(* Logix 5000 project; controller CLASE_1 Emulate 5570 rev 28.11; software revision 28.02; part 12 of 15 *)
(* tags used below, declared in another part *)
   Inp_SpeedFdbk : REAL;   // Speed Feedbak in Drive Units (typ. 0-32767 = 0 to max freq.)
   Inp_Datalink : REAL;   // Auxiliary Signal (datalink) Input in Drive (raw) Units
   Inp_Ready : BOOL;   // 1=Drive is ready to run
   Inp_Running : BOOL;   // 1=Drive is Running (active)
   Inp_CommandDir : BOOL;   // 1=Drive is commanded Forward, 0=Drive is commanded Reverse
   Inp_ActualDir : BOOL;   // 1=Drive is running Forward, 0=Drive is running Reverse
   Inp_Accelerating : BOOL;   // 1=Drive is accelerating
   Inp_Decelerating : BOOL;   // 1=Drive is decelerating
   Inp_Alarm : BOOL;   // 1=Drive has an Alarm Condition (see drive display or manual)
   Inp_Faulted : BOOL;   // 1=Drive has Faulted (see drive display or manual)
   Inp_AtSpeed : BOOL;   // 1=Drive is at commanded speed
   Inp_FwdPermOK : BOOL;   // 1=Permissives OK, drive can start Forward
   Inp_FwdNBPermOK : BOOL;   // 1=Non-Bypassable Permissives OK, drive can start Forward
   Inp_RevPermOK : BOOL;   // 1=Permissives OK, drive can start Reverse
   Inp_RevNBPermOK : BOOL;   // 1=Non-Bypassable Permissives OK, motor can start Reverse
   Inp_IntlkOK : BOOL;   // 1=Interlocks OK, drive can start/run
   Inp_NBIntlkOK : BOOL;   // 1=Non-Bypassable Interlocks OK, drive can start/run
   Inp_IOFault : BOOL;   // Input Communication Status 0=OK, 1=fail
   Inp_Sim : BOOL;   // 1=Simulate working drive; 0=Start/Stop/ Monitor actual drive
   Inp_OvrdCmd : SINT;   // Override Mode Command: 0=None, 1=Stop, 2=Start Fwd 3=Start Rev
   Inp_Reset : BOOL;   // 1=Reset drive fault conditions and latched Alarms
   Cfg_HasReverse : BOOL;   // 1=Drive can be run reverse, 0=Forward only
   Cfg_AllowLocal : BOOL;   // 1=Allow Local Start/Stop without alarm, 0=Start/Stop from HMI/prog only
   Cfg_HasRunFdbk : BOOL;   // 1=Drive provides feedback signal on Inp_Running when running
   Cfg_UseRunFdbk : BOOL;   // 1=Drive run feedback should be used for failure checking
   Cfg_HasSpeedFdbk : BOOL;   // 1=Drive provides speed feedback on Inp_SpeedFdbk
   Cfg_UseSpeedFdbk : BOOL;   // 1=Drive speed determines running state, 0=state determined by drive Active input bit
   Cfg_HasInpDatalink : BOOL;   // 1=A signal is connected to Inp_Datalink
   Cfg_PCmdClear : ALIAS FOR Mode.Cfg_PCmdClear;
   Cfg_OperStopPrio : BOOL;   // 1=OCmd_Stop has priority, accepted any time, 0=OCmd_Stop only in Oper, Maint Mode.
   Cfg_OCmdResets : BOOL;   // 1=New Oper drive cmd. resets fault, 0=reset req'd to clear fault
   Cfg_OvrdPermIntlk : BOOL;   // 1=Override ignores Bypassable Perm/ Intlk; 0=always use Perm/Intlk
   Cfg_ShedOnFailToStart : BOOL;   // 1=Stop Motor and Alarm on Fail to Start; 0=Alarm only on Fail to Start
   Cfg_ShedOnIOFault : BOOL;   // 1=Stop Motor and Alarm on I/O Fault; 0=Alarm only on I/O Fault
   Cfg_SimScaleEU : BOOL;   // 1=In simulation, scale Speed Ref EU to Speed Fdbk EU
   Cfg_SimScaleRaw : BOOL;   // 1=In simulation, scale Speed Ref EU to raw, then raw to Speed Fdbk EU
   Cfg_MaxSpdRef : REAL;   // Maximum Speed Reference in EU (for limiting)
   Cfg_SpeedRefRawMin : REAL;   // Speed Reference Minimum in Drive (raw) Units (for scaling)
   Cfg_SpeedRefRawMax : REAL;   // Speed Reference Maximum in Drive (raw) Units (for scaling)
   Cfg_SpeedRefEUMin : REAL;   // Speed Reference Minimum in Engineering Units (for scaling)
   Cfg_SpeedRefEUMax : REAL;   // Speed Reference Maximum in Engineering Units (for scaling)
   Cfg_SpeedFdbkRawMin : REAL;   // Speed Feedback Minimum in Drive (raw) Units (for scaling)
   Cfg_SpeedFdbkRawMax : REAL;   // Speed Feedback Maximum in Drive (raw) Units (for scaling)
   Cfg_SpeedFdbkEUMin : REAL;   // Speed Feedback Minimum in Engineering Units (for scaling)
   Cfg_SpeedFdbkEUMax : REAL;   // Speed Feedback Maximum in Engineering Units (for scaling)
   Cfg_InpDatalinkRawMin : REAL;   // Input Datalink Minimum in Drive (raw) Units (for scaling)
   Cfg_InpDatalinkRawMax : REAL;   // Input Datalink Maximum in Drive (raw) Units (for scaling)
   Cfg_InpDatalinkEUMin : REAL;   // Input Datalink Minimum in Engineering Units (for scaling)
   Cfg_InpDatalinkEUMax : REAL;   // Input Datalink Maximum in Engineering Units (for scaling)
   Cfg_SimRampT : DINT;   // Time to ramp speed fdbk when in Simulation (sec)
   Cfg_OperKeep : SINT;   // Oper keeps control in Prog Mode: .0=Reference, .1=Start/Stop, .2=Fwd/Rev, .3=OutDatalink
   Cfg_ProgKeep : SINT;   // Prog keeps control in Oper Mode: .0=Reference, .1=Start/Stop, .2=Fwd/Rev, .3=OutDatalink
   PCmd_Start : BOOL;   // Program Command to Start Drive
   PCmd_Stop : BOOL;   // Program Command to Stop Drive
   PCmd_Fwd : BOOL;   // Program Command to set direction to Fowrard
   PCmd_Rev : BOOL;   // Program Command to set direction to Reverse
   PCmd_Reset : BOOL;   // Program Command to Reset drive fault and all Alarms requiring Reset
   PCmd_FailToStartAck : ALIAS FOR FailToStart.PCmd_Ack;   // Program Command to Acknowledge Fail to Start Alarm
   PCmd_FailToStopAck : ALIAS FOR FailToStop.PCmd_Ack;   // Program Command to Acknowledge Fail to Stop Alarm
   PCmd_IntlkTripAck : ALIAS FOR IntlkTrip.PCmd_Ack;   // Program Command to Acknowledge Interlock Trip Alarm
   PCmd_DriveFaultAck : ALIAS FOR DriveFault.PCmd_Ack;   // Program Command to Acknowledge Drive Fault Alarm
   PCmd_IOFaultAck : ALIAS FOR IOFault.PCmd_Ack;   // Program Command to Acknowledge I/O Fault Alarm
   OCmd_Start : BOOL;   // Operator Command to Start Drive
   OCmd_Stop : BOOL;   // Operator Command to Stop Drive
   OCmd_Jog : BOOL;   // Operator Command to Jog Drive (not cleared by P_VSD!)
   OCmd_Fwd : BOOL;   // Operator Command to set direction to Forward
   OCmd_Rev : BOOL;   // Operator Command to set direction to Reverse
   OCmd_Bypass : BOOL;   // Operator Command to Bypass all Bypassable Interlocks and Permissives
   OCmd_Check : BOOL;   // Operator Command to Check (not bypass) all Interlocks and Permissives
   MCmd_Disable : BOOL;   // Maintenance Command to Disable Drive
   MCmd_Enable : BOOL;   // Maintenance Command to Enable (allow to run) Drive
   OCmd_Reset : BOOL;   // Operator Command to Reset all Alarms requiring Reset
   OCmd_ResetAckAll : BOOL;   // Operator Command to Reset all Alarms and latched Shed conditions
   Out_Stop : BOOL;   // 1=Stop Drive, 0=drive left in current state
   Out_Start : BOOL;   // 1=Start Drive, 0=drive left in current state
   Out_ClearFault : BOOL;   // 1=Attempt to clear Drive Fault
   Val_SpeedFdbk : REAL;   // Speed Feedback (actual) from drive
   Val_InpDatalink : REAL;   // Input Datalink value from drive
   Val_Fdbk : SINT;   // Device Feedback 0=Stopped, 1=Running Fwd 2=Running Rev 3=Accelerating 4=Decelerating
   Sts_Starting : BOOL;   // 1=Drive requested to run and awaiting run feedback
   Sts_Running : BOOL;   // 1=Drive requested to run and is confirmed running
   Sts_CommandDir : BOOL;   // 1=Drive commanded to Forward, 0=Reverse
   Sts_ActualDir : BOOL;   // 1=Drive Actual direction is Forward, 0=Reverse
   Sts_Accel : BOOL;   // 1=Drive is Accelerating
   Sts_Decel : BOOL;   // 1=Drive is Decelerating
   Sts_NotReady : BOOL;   // 1=Drive is Not Ready (cannot be started) Check alarms, stops, faults
   Sts_Alarm : BOOL;   // 1=Drive has an Alarm (see drive display or manual)
   Sts_AtSpeed : BOOL;   // 1=Drive is running at reference speed
   Sts_Available : BOOL;   // 1=Drive available for control by automation (Prog)
   Sts_Bypass : BOOL;   // 1=Bypassable Interlocks and Permissives are Bypassed
   Sts_BypActive : BOOL;   // 1=Bypassing Active (Bypassed or Maintenance)
   Sts_Disabled : BOOL;   // 1=Drive is Disabled
   Sts_NotRdy : BOOL;   // 1=Device Not Ready, see detail bits for reason
   Nrdy_Disabled : BOOL;   // 1=Device Not Ready: Device Disabled by Maintenance
   Nrdy_CfgErr : BOOL;   // 1=Device Not Ready: Configuration Error
   Nrdy_Intlk : BOOL;   // 1=Device Not Ready: Interlock Not OK
   Nrdy_Perm : BOOL;   // 1=Device Not Ready: Permissive Not OK
   Nrdy_OperPrio : BOOL;   // 1=Device Not Ready: Operator State 0 Priority Command Requires Reset
   Nrdy_Fail : BOOL;   // 1=Device Not Ready: Device Failure (Shed Requires Reset)
   Nrdy_IOFault : BOOL;   // 1=Device Not Ready: I/O Fault (Shed Requires Reset)
   Nrdy_Trip : BOOL;   // 1=Device not Ready: Deivce Tripped (Drive Fault)
   Nrdy_DriveNR : BOOL;   // 1=Device Note Ready: Drive Not Ready
   Nrdy_NoMode : BOOL;   // 1=Device Not Ready: Device Logic Disabled / NO Mode
   Sts_MaintByp : BOOL;   // 1=A Maintenance Bypass is Active, display icon
   Sts_Err : BOOL;   // 1=Error in Config: see detail bits for reason
   Err_FdbkRaw : BOOL;   // 1=Erron in Config: Speed Fdbk Raw Min = Max
   Err_FdbkEU : BOOL;   // 1=Error in Config: Speed Fdbk EU Min = Max
   Err_RefEU : BOOL;   // 1=Error in Config: Speed Ref EU Min = Max
   Err_InpDLEU : BOOL;   // 1=Error in Config: Input Datalink EU Min = Max
   Sts_Hand : ALIAS FOR Mode.Sts_Hand;
   Sts_Maint : ALIAS FOR Mode.Sts_Maint;
   Sts_Ovrd : ALIAS FOR Mode.Sts_Ovrd;
   Sts_Prog : ALIAS FOR Mode.Sts_Prog;
   Sts_Oper : ALIAS FOR Mode.Sts_Oper;
   Sts_FailToStart : ALIAS FOR FailToStart.Inp;   // 1=Drive Failed to Start (One-Shot)
   Sts_FailToStop : ALIAS FOR FailToStop.Inp;   // 1=Drive Failed to Stop
   Sts_IntlkTrip : ALIAS FOR IntlkTrip.Inp;   // 1=Drive was stopped by an Interlock NOT OK (One-Shot)
   Sts_DriveFault : ALIAS FOR DriveFault.Inp;   // 1=Drive Fault (see drive display or manual)
   Sts_IOFault : ALIAS FOR IOFault.Inp;   // I/O Comm Fault Status (0=OK, 1=Bad)
   Rdy_Fwd : BOOL;   // 1=Ready to receive OCmd_Fwd (enabled HMI button)
   Rdy_Rev : BOOL;   // 1=Ready to receive OCmd_Rev (enables HMI button)
   Rdy_Bypass : BOOL;   // 1=Ready to receive OCmd_Bypass (enables HMI button)
   Rdy_Check : BOOL;   // 1=Ready to receive OCmd_Check (enables HMI button)
   Rdy_Disable : BOOL;   // 1=Ready to receive MCmd_Disable (enables HMI button)
   Rdy_Enable : BOOL;   // 1=Ready to receive MCmd_Enable (enables HMI button)
   P_VSD : BOOL;   // Unique Parameter Name for auto - discovery
   Mode : P_Mode;   // Drive Mode Selection
   IOFault : P_Alarm;   // I/O Fault Alarm
   IntlkTrip : P_Alarm;   // Interlock Trip Alarm
   FailToStop : P_Alarm;   // Drive Failed to Stop Alarm
   FailToStart : P_Alarm;   // Drive Failed to Start Alarm
   Wrk_Run : BOOL;   // 1=Drive should be "running", 0=should be "stopped"
   Wrk_StartRetrigT : TIMER;   // Time to pulse start output on start command retrigger (Maint)
   Wrk_StopRetrigT : TIMER;   // Time to pulse stop output on stop command retrigger (Maint)
   Wrk_RunFdbk : BOOL;   // Run Feedback based on mode, simulation, etc. 1=running
   Wrk_Bypass : BOOL;   // Internal Bypassable Permissives and Interlocks are Bypassed flag
   Wrk_Disabled : BOOL;   // Internal Drive is Disabled
   DriveFault : P_Alarm;   // Drive Faulted Alarm
   Wrk_SpeedRef : REAL;   // Working copy of Speed Reference (for limiting)
   Wrk_Rev : BOOL;   // Working (internal) Direction 1=Reverse 0=Forward (default)
   Wrk_Jog : BOOL;   // 1=Jog Drive, 0=Drive not jogging
   Wrk_ResetT : TIMER;   // Reset Output Pulse Timer
   Wrk_ResetONS : BOOL;   // One-Shot to fire Reset Timer to ensure min. output ON time.
   Wrk_StopT : TIMER;   // Stop Check Timer (for Fail to Stop)
   Wrk_StartT : TIMER;   // Start Check Timer (for Fail to Start)
   Wrk_Retrigger : BOOL;   // Maint Start issued while running or Stop while stopped
   Wrk_Step : REAL;   // Amount to change simulated Speed Fdbk this scan (ramp)
   Wrk_ScanTime : REAL;   // Seconds since previous scan
   Wrk_SimFdbkTgt : REAL;   // Speed Ref converted to Speed Fdbk units for simulation: target speed fdbk
   Wrk_JogT : TIMER;   // Jog Timer
   Wrk_SimScaleEUONS : BOOL;   // Cfg_SimScaleEU became true this scan
   Wrk_SimScaleRawONS : BOOL;   // Cfg_SimScaleRaw became true this scan
   Wrk_NotRdyONS : BOOL;   // Assert Stop on One-Shot of Sts_NotRdy
   Wrk_NotRdy : BOOL;   // Device Not Ready conditions excluding shed latches
   Wrk_StartInhT : TIMER;   // Local Start Inhibit Timer
   Wrk_StopInhT : TIMER;   // Local Stop Inhibit Timer
   Wrk_Hand : BOOL;   // Perform Hand Mode alignment with actual device state
   Wrk_RevCmdRcvd : BOOL;   // A Reverse direction command was received this scan.
   Wrk_FwdCmdRcvd : BOOL;   // A Forward direction command was received this scan
(* P_VSD, continued *)

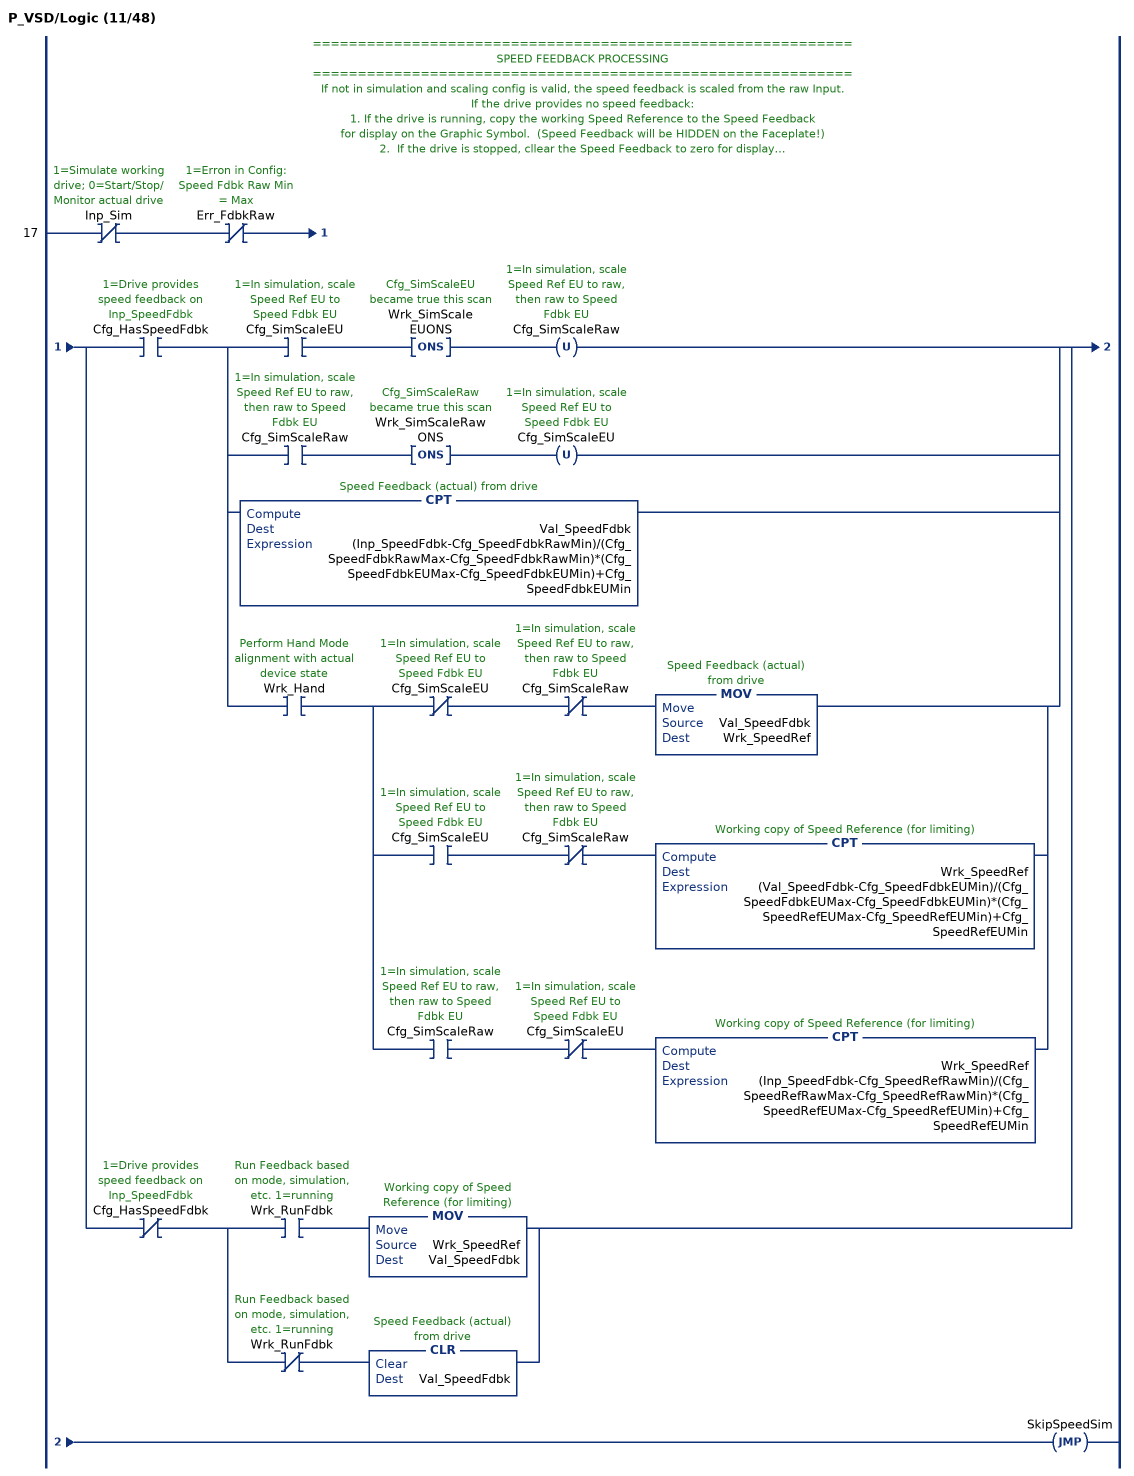
   // ============================================================
   // SPEED FEEDBACK PROCESSING
   // ============================================================
   // If not in simulation and scaling config is valid, the speed feedback is scaled from the raw Input.
   // If the drive provides no speed feedback:
   // 1. If the drive is running, copy the working Speed Reference to the Speed Feedback
   // for display on the Graphic Symbol.  (Speed Feedback will be HIDDEN on the Faceplate!)
   // 2.  If the drive is stopped, cllear the Speed Feedback to zero for display.
   // #####  V3.0-00  2013-06-30:  Added Cfg_HasSpeedFdbk  #####
   // #####  V3.0-05  2014-05-20:  Modified to prevent both Simulation  #####
   // #####  scaling bits from being set at the same time.  #####
   // #####  V3.1-04 Patch01  2015-09-25:  Added logic for Cfg_HasSpeedFdbk = 0  #####
   // #####  V3.5-04  2016-09-30:  Modified to ensure instruction  #####
   // #####  aligns with actual state of the drive on transistion from Sim to Real.  #####
   17: XIO(Inp_Sim)XIO(Err_FdbkRaw)[XIC(Cfg_HasSpeedFdbk) [XIC(Cfg_SimScaleEU) ONS(Wrk_SimScaleEUONS) OTU(Cfg_SimScaleRaw) ,XIC(Cfg_SimScaleRaw) ONS(Wrk_SimScaleRawONS) OTU(Cfg_SimScaleEU) ,CPT(Val_SpeedFdbk,(Inp_SpeedFdbk-Cfg_SpeedFdbkRawMin)/(Cfg_SpeedFdbkRawMax-Cfg_SpeedFdbkRawMin)*(Cfg_SpeedFdbkEUMax-Cfg_SpeedFdbkEUMin)+Cfg_SpeedFdbkEUMin) ,XIC(Wrk_Hand) [XIO(Cfg_SimScaleEU) XIO(Cfg_SimScaleRaw) MOV(Val_SpeedFdbk,Wrk_SpeedRef) ,XIC(Cfg_SimScaleEU) XIO(Cfg_SimScaleRaw) CPT(Wrk_SpeedRef,(Val_SpeedFdbk-Cfg_SpeedFdbkEUMin)/(Cfg_SpeedFdbkEUMax-Cfg_SpeedFdbkEUMin)*(Cfg_SpeedRefEUMax-Cfg_SpeedRefEUMin)+Cfg_SpeedRefEUMin) ,XIC(Cfg_SimScaleRaw) XIO(Cfg_SimScaleEU) CPT(Wrk_SpeedRef,(Inp_SpeedFdbk-Cfg_SpeedRefRawMin)/(Cfg_SpeedRefRawMax-Cfg_SpeedRefRawMin)*(Cfg_SpeedRefEUMax-Cfg_SpeedRefEUMin)+Cfg_SpeedRefEUMin) ] ] ,XIO(Cfg_HasSpeedFdbk) [XIC(Wrk_RunFdbk) MOV(Wrk_SpeedRef,Val_SpeedFdbk) ,XIO(Wrk_RunFdbk) CLR(Val_SpeedFdbk) ] ]JMP(SkipSpeedSim);
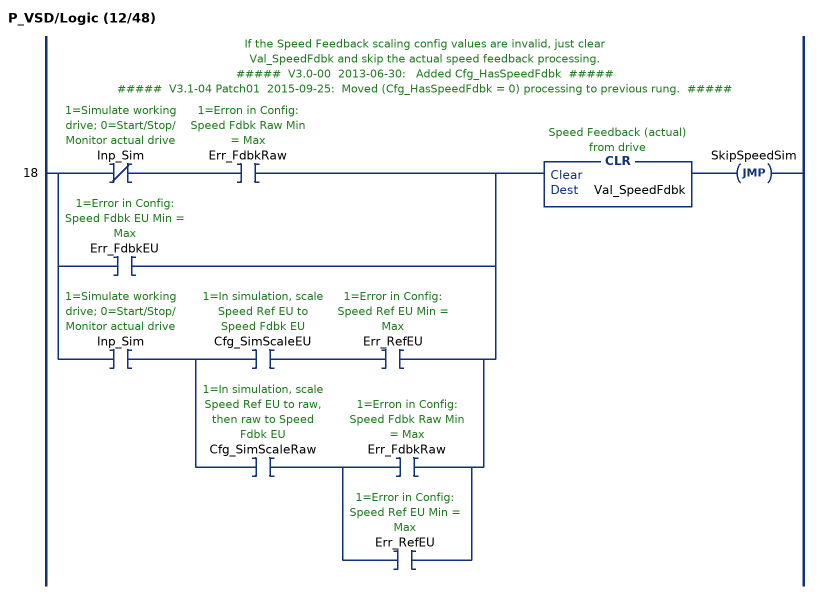
   // If the Speed Feedback scaling config values are invalid, just clear
   // Val_SpeedFdbk and skip the actual speed feedback processing.
   // #####  V3.0-00  2013-06-30:   Added Cfg_HasSpeedFdbk  #####
   // #####  V3.1-04 Patch01  2015-09-25:  Moved (Cfg_HasSpeedFdbk = 0) processing to previous rung.  #####
   18: [XIO(Inp_Sim) XIC(Err_FdbkRaw) ,XIC(Err_FdbkEU) ,XIC(Inp_Sim) [XIC(Cfg_SimScaleEU) XIC(Err_RefEU) ,XIC(Cfg_SimScaleRaw) [XIC(Err_FdbkRaw) ,XIC(Err_RefEU) ] ] ]CLR(Val_SpeedFdbk)JMP(SkipSpeedSim);
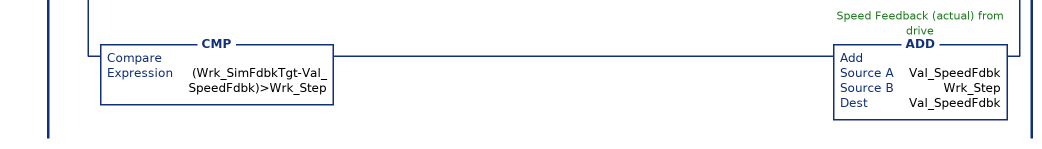
   // If in simulation, simulate accel/decel.
   19: XIC(Inp_Sim)[[XIC(Wrk_Run) ,XIC(Wrk_Jog) ] [XIO(Cfg_SimScaleEU) XIO(Cfg_SimScaleRaw) MOV(Wrk_SpeedRef,Wrk_SimFdbkTgt) ,[XIC(Cfg_SimScaleEU) XIO(Cfg_SimScaleRaw) CPT(Wrk_SimFdbkTgt,(Wrk_SpeedRef-Cfg_SpeedRefEUMin)/(Cfg_SpeedRefEUMax-Cfg_SpeedRefEUMin)*(Cfg_SpeedFdbkEUMax-Cfg_SpeedFdbkEUMin)+Cfg_SpeedFdbkEUMin) ,XIC(Cfg_SimScaleRaw) [CPT(Wrk_SimFdbkTgt,(Wrk_SpeedRef-Cfg_SpeedRefEUMin)/(Cfg_SpeedRefEUMax-Cfg_SpeedRefEUMin)*(Cfg_SpeedRefRawMax-Cfg_SpeedRefRawMin)+Cfg_SpeedRefRawMin) ,CPT(Wrk_SimFdbkTgt,(Wrk_SimFdbkTgt-Cfg_SpeedFdbkRawMin)/(Cfg_SpeedFdbkRawMax-Cfg_SpeedFdbkRawMin)*(Cfg_SpeedFdbkEUMax-Cfg_SpeedFdbkEUMin)+Cfg_SpeedFdbkEUMin) ] ] ] ,[XIO(Wrk_Run) XIO(Wrk_Jog) ,XIO(Wrk_Rev) XIO(Sts_ActualDir) ,XIC(Wrk_Rev) XIC(Sts_ActualDir) ] CLR(Wrk_SimFdbkTgt) ,GRT(Cfg_SimRampT,0) [CPT(Wrk_Step,Cfg_MaxSpdRef/Cfg_SimRampT*Wrk_ScanTime) ,XIC(Cfg_SimScaleEU) XIO(Cfg_SimScaleRaw) CPT(Wrk_Step,(Wrk_Step-Cfg_SpeedRefEUMin)/(Cfg_SpeedRefEUMax-Cfg_SpeedRefEUMin)*(Cfg_SpeedFdbkEUMax-Cfg_SpeedFdbkEUMin)+Cfg_SpeedFdbkEUMin) ,XIC(Cfg_SimScaleRaw) [CPT(Wrk_Step,(Wrk_Step-Cfg_SpeedRefEUMin)/(Cfg_SpeedRefEUMax-Cfg_SpeedRefEUMin)*(Cfg_SpeedRefRawMax-Cfg_SpeedRefRawMin)+Cfg_SpeedRefRawMin) ,CPT(Wrk_Step,(Wrk_Step-Cfg_SpeedFdbkRawMin)/(Cfg_SpeedFdbkRawMax-Cfg_SpeedFdbkRawMin)*(Cfg_SpeedFdbkEUMax-Cfg_SpeedFdbkEUMin)+Cfg_SpeedFdbkEUMin) ] ] ,LEQ(Cfg_SimRampT,0) MOV(1.50000000e+038,Wrk_Step) ,CMP(ABS(Val_SpeedFdbk-Wrk_SimFdbkTgt)<=Wrk_Step) MOV(Wrk_SimFdbkTgt,Val_SpeedFdbk) ,CMP((Val_SpeedFdbk-Wrk_SimFdbkTgt)>Wrk_Step) SUB(Val_SpeedFdbk,Wrk_Step,Val_SpeedFdbk) ,CMP((Wrk_SimFdbkTgt-Val_SpeedFdbk)>Wrk_Step) ADD(Val_SpeedFdbk,Wrk_Step,Val_SpeedFdbk) ];
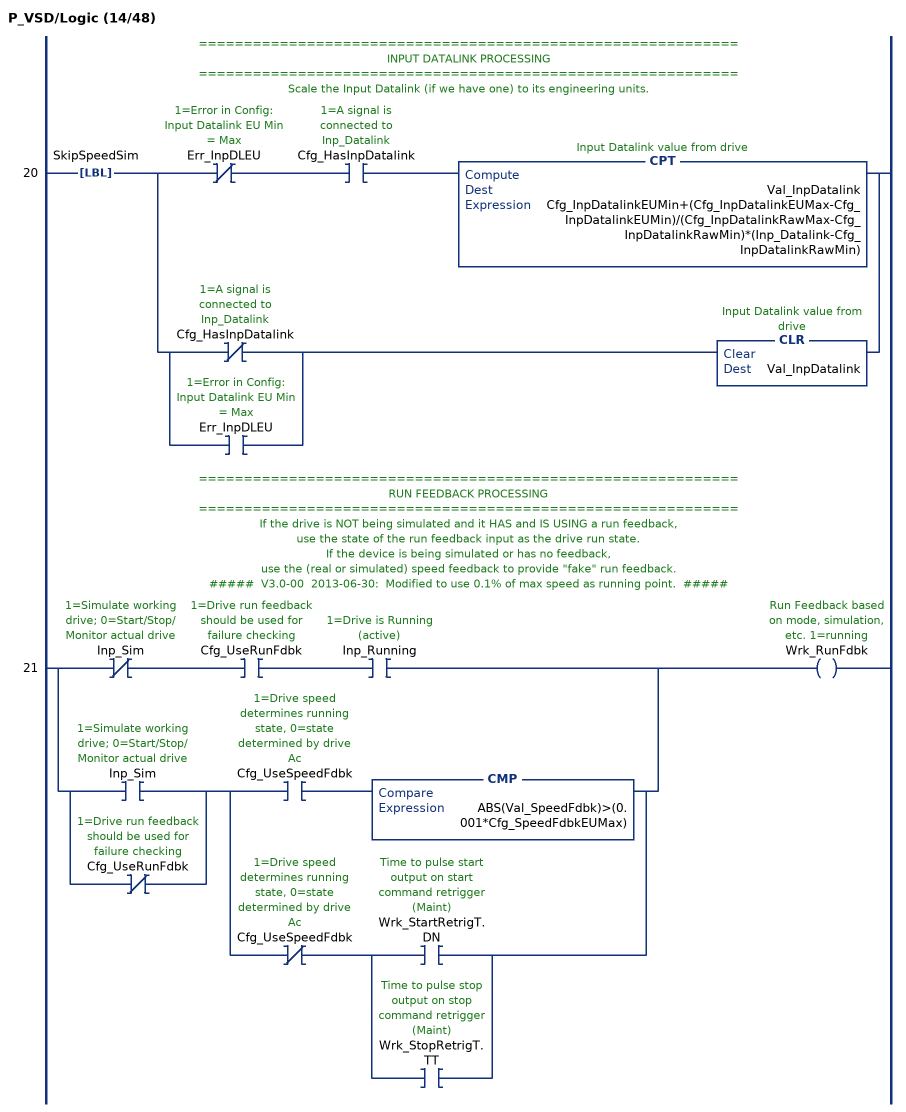
   // ============================================================
   // INPUT DATALINK PROCESSING
   // ============================================================
   // Scale the Input Datalink (if we have one) to its engineering units.
   20: LBL(SkipSpeedSim)[XIO(Err_InpDLEU) XIC(Cfg_HasInpDatalink) CPT(Val_InpDatalink,Cfg_InpDatalinkEUMin+(Cfg_InpDatalinkEUMax-Cfg_InpDatalinkEUMin)/(Cfg_InpDatalinkRawMax-Cfg_InpDatalinkRawMin)*(Inp_Datalink-Cfg_InpDatalinkRawMin)) ,[XIO(Cfg_HasInpDatalink) ,XIC(Err_InpDLEU) ] CLR(Val_InpDatalink) ];
   // ============================================================
   // RUN FEEDBACK PROCESSING
   // ============================================================
   // If the drive is NOT being simulated and it HAS and IS USING a run feedback,
   // use the state of the run feedback input as the drive run state.
   // If the device is being simulated or has no feedback,
   // use the (real or simulated) speed feedback to provide "fake" run feedback.
   // #####  V3.0-00  2013-06-30:  Modified to use 0.1% of max speed as running point.  #####
   21: [XIO(Inp_Sim) XIC(Cfg_UseRunFdbk) XIC(Inp_Running) ,[XIC(Inp_Sim) ,XIO(Cfg_UseRunFdbk) ] [XIC(Cfg_UseSpeedFdbk) CMP(ABS(Val_SpeedFdbk)>(0.001*Cfg_SpeedFdbkEUMax)) ,XIO(Cfg_UseSpeedFdbk) [XIC(Wrk_StartRetrigT.DN) ,XIC(Wrk_StopRetrigT.TT) ] ] ]OTE(Wrk_RunFdbk);
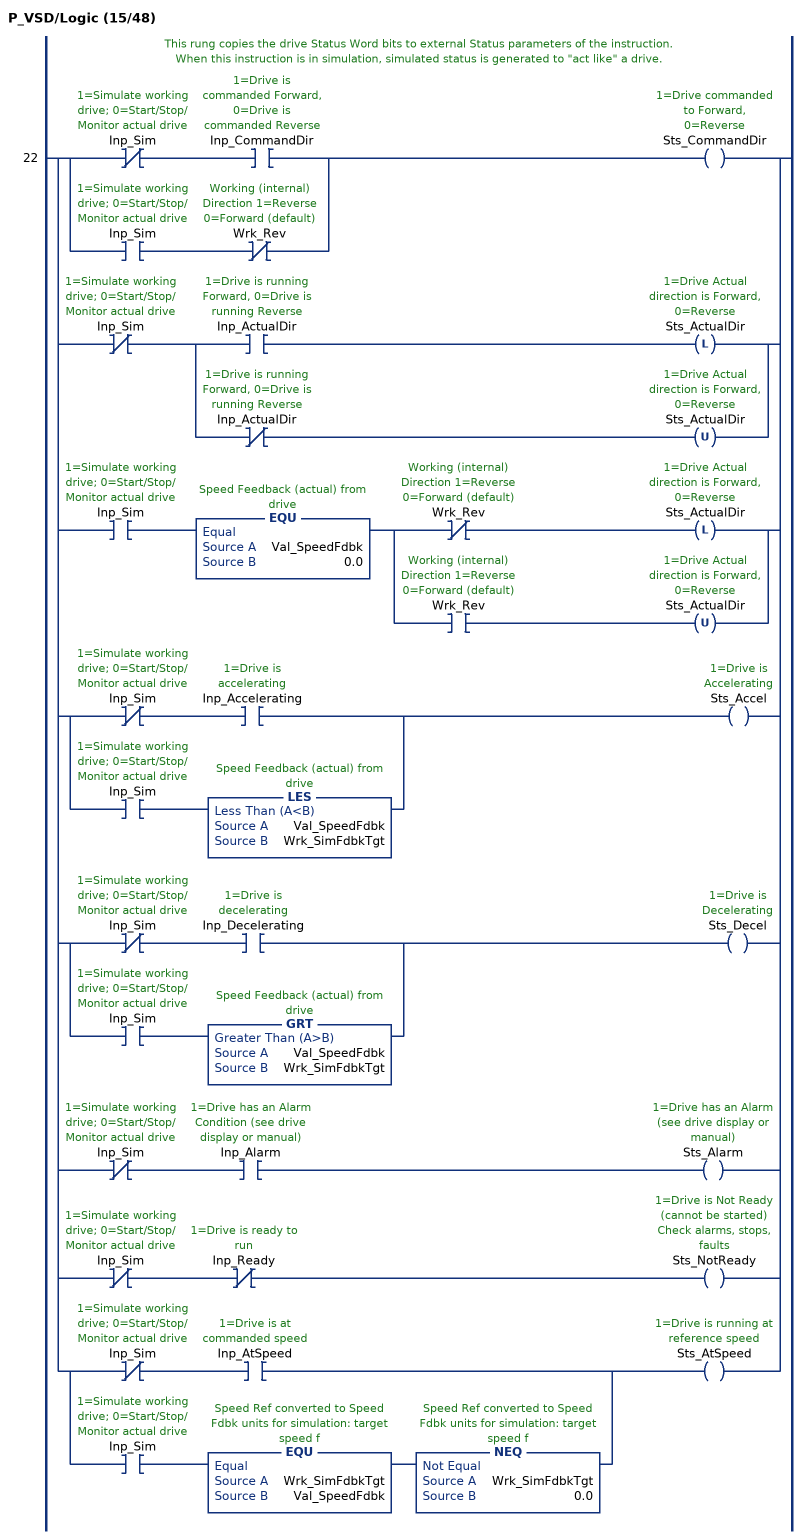
   // This rung copies the drive Status Word bits to external Status parameters of the instruction.
   // When this instruction is in simulation, simulated status is generated to "act like" a drive.
   22: [[XIO(Inp_Sim) XIC(Inp_CommandDir) ,XIC(Inp_Sim) XIO(Wrk_Rev) ] OTE(Sts_CommandDir) ,[XIO(Inp_Sim) [XIC(Inp_ActualDir) OTL(Sts_ActualDir) ,XIO(Inp_ActualDir) OTU(Sts_ActualDir) ] ,XIC(Inp_Sim) EQU(Val_SpeedFdbk,0.0) [XIO(Wrk_Rev) OTL(Sts_ActualDir) ,XIC(Wrk_Rev) OTU(Sts_ActualDir) ] ] ,[XIO(Inp_Sim) XIC(Inp_Accelerating) ,XIC(Inp_Sim) LES(Val_SpeedFdbk,Wrk_SimFdbkTgt) ] OTE(Sts_Accel) ,[XIO(Inp_Sim) XIC(Inp_Decelerating) ,XIC(Inp_Sim) GRT(Val_SpeedFdbk,Wrk_SimFdbkTgt) ] OTE(Sts_Decel) ,XIO(Inp_Sim) XIC(Inp_Alarm) OTE(Sts_Alarm) ,XIO(Inp_Sim) XIO(Inp_Ready) OTE(Sts_NotReady) ,[XIO(Inp_Sim) XIC(Inp_AtSpeed) ,XIC(Inp_Sim) EQU(Wrk_SimFdbkTgt,Val_SpeedFdbk) NEQ(Wrk_SimFdbkTgt,0.0) ] OTE(Sts_AtSpeed) ];
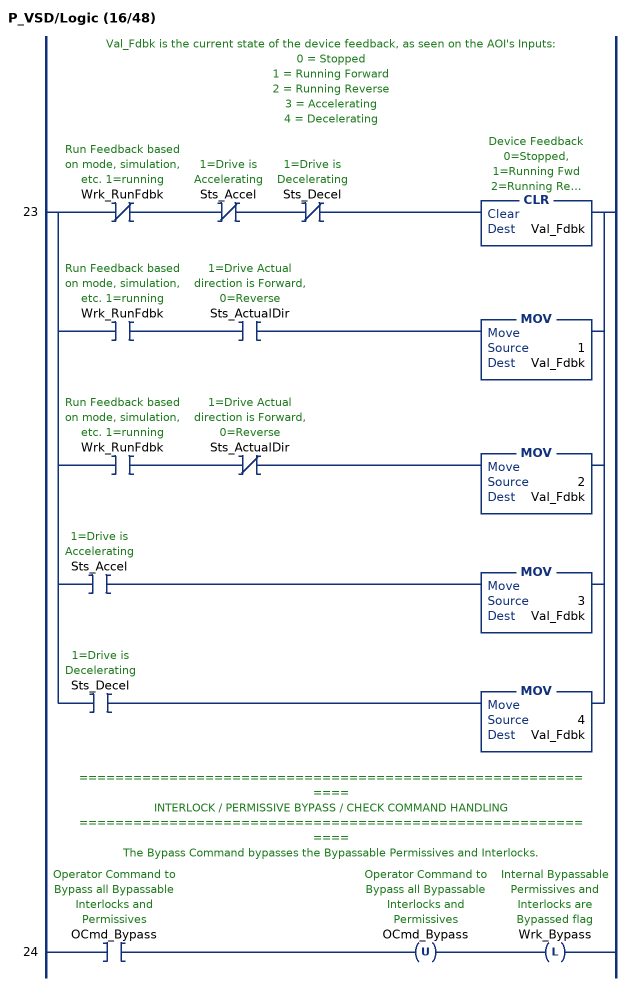
   // Val_Fdbk is the current state of the device feedback, as seen on the AOI's Inputs:
   // 0 = Stopped
   // 1 = Running Forward
   // 2 = Running Reverse
   // 3 = Accelerating
   // 4 = Decelerating
   23: [XIO(Wrk_RunFdbk) XIO(Sts_Accel) XIO(Sts_Decel) CLR(Val_Fdbk) ,XIC(Wrk_RunFdbk) XIC(Sts_ActualDir) MOV(1,Val_Fdbk) ,XIC(Wrk_RunFdbk) XIO(Sts_ActualDir) MOV(2,Val_Fdbk) ,XIC(Sts_Accel) MOV(3,Val_Fdbk) ,XIC(Sts_Decel) MOV(4,Val_Fdbk) ];
   // ============================================================
   // INTERLOCK / PERMISSIVE BYPASS / CHECK COMMAND HANDLING
   // ============================================================
   // The Bypass Command bypasses the Bypassable Permissives and Interlocks.
   24: XIC(OCmd_Bypass)OTU(OCmd_Bypass)OTL(Wrk_Bypass);
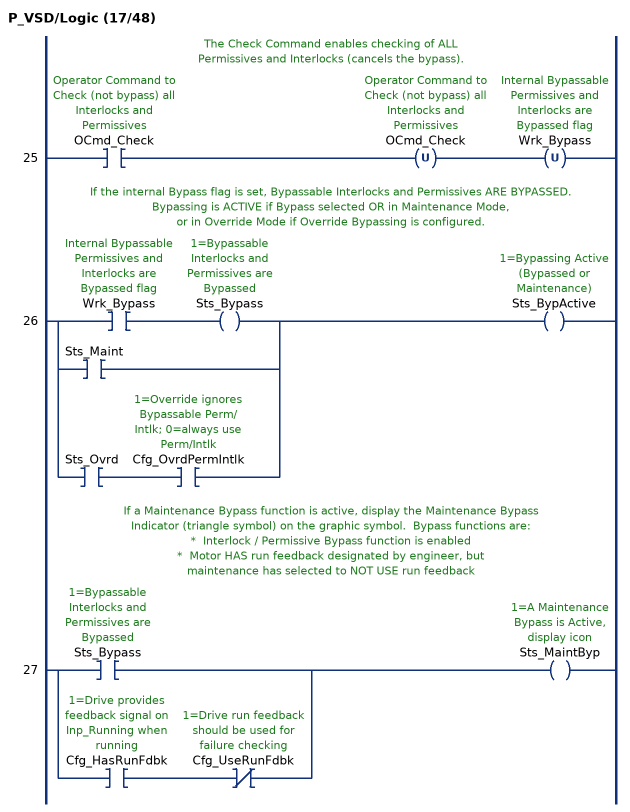
   // The Check Command enables checking of ALL
   // Permissives and Interlocks (cancels the bypass).
   25: XIC(OCmd_Check)OTU(OCmd_Check)OTU(Wrk_Bypass);
   // If the internal Bypass flag is set, Bypassable Interlocks and Permissives ARE BYPASSED.
   // Bypassing is ACTIVE if Bypass selected OR in Maintenance Mode,
   // or in Override Mode if Override Bypassing is configured.
   26: [XIC(Wrk_Bypass) OTE(Sts_Bypass) ,XIC(Sts_Maint) ,XIC(Sts_Ovrd) XIC(Cfg_OvrdPermIntlk) ]OTE(Sts_BypActive);
   // If a Maintenance Bypass function is active, display the Maintenance Bypass
   // Indicator (triangle symbol) on the graphic symbol.  Bypass functions are:
   // *  Interlock / Permissive Bypass function is enabled
   // *  Motor HAS run feedback designated by engineer, but
   // maintenance has selected to NOT USE run feedback
   27: [XIC(Sts_Bypass) ,XIC(Cfg_HasRunFdbk) XIO(Cfg_UseRunFdbk) ]OTE(Sts_MaintByp);
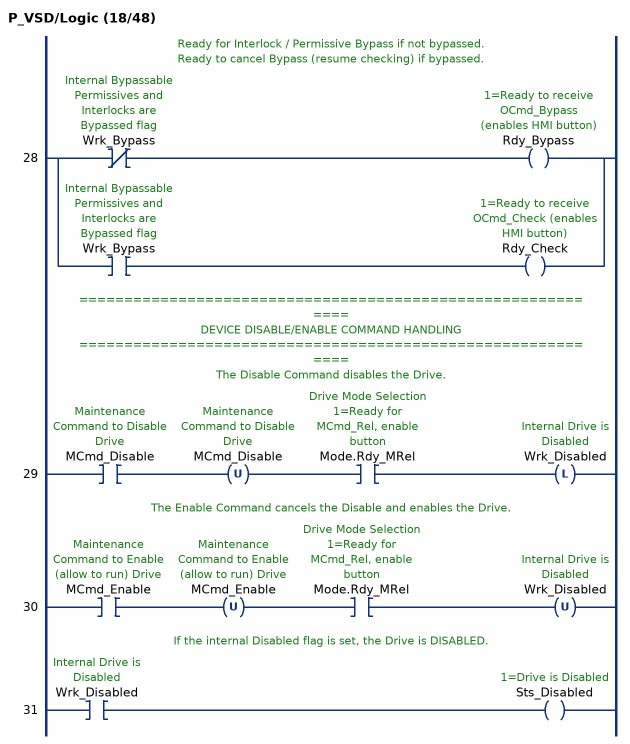
   // Ready for Interlock / Permissive Bypass if not bypassed.
   // Ready to cancel Bypass (resume checking) if bypassed.
   28: [XIO(Wrk_Bypass) OTE(Rdy_Bypass) ,XIC(Wrk_Bypass) OTE(Rdy_Check) ];
   // ============================================================
   // DEVICE DISABLE/ENABLE COMMAND HANDLING
   // ============================================================
   // The Disable Command disables the Drive.
   29: XIC(MCmd_Disable)OTU(MCmd_Disable)XIC(Mode.Rdy_MRel)OTL(Wrk_Disabled);
   // The Enable Command cancels the Disable and enables the Drive.
   30: XIC(MCmd_Enable)OTU(MCmd_Enable)XIC(Mode.Rdy_MRel)OTU(Wrk_Disabled);
   // If the internal Disabled flag is set, the Drive is DISABLED.
   31: XIC(Wrk_Disabled)OTE(Sts_Disabled);
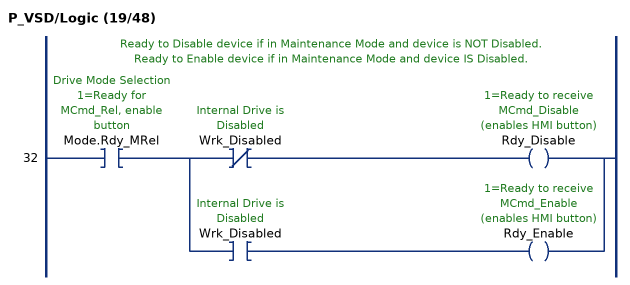
   // Ready to Disable device if in Maintenance Mode and device is NOT Disabled.
   // Ready to Enable device if in Maintenance Mode and device IS Disabled.
   32: XIC(Mode.Rdy_MRel)[XIO(Wrk_Disabled) OTE(Rdy_Disable) ,XIC(Wrk_Disabled) OTE(Rdy_Enable) ];
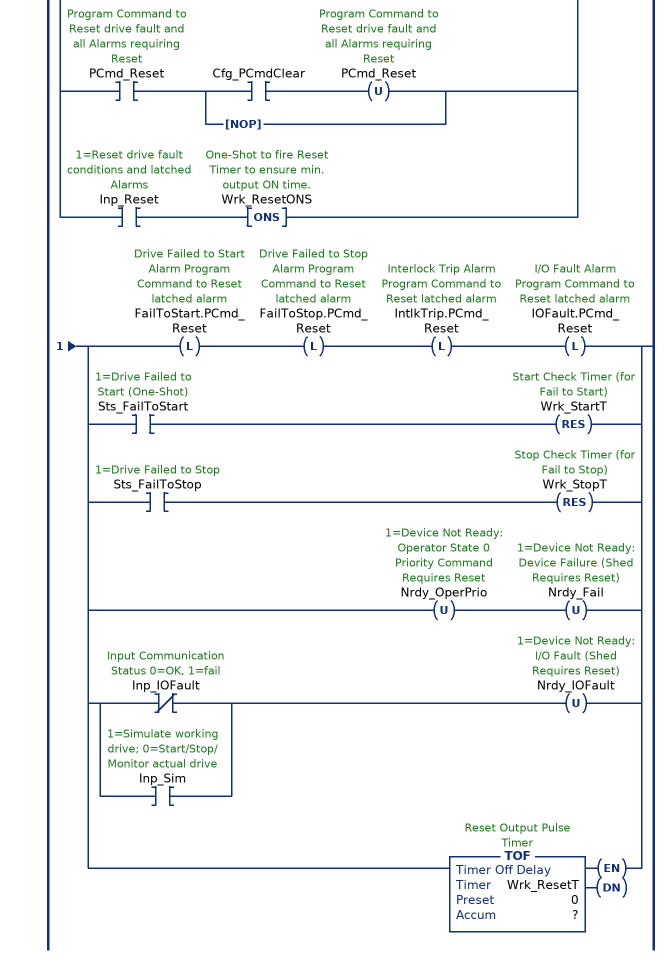
   // ============================================================
   // ALARM RESET COMMAND HANDLING
   // ============================================================
   // This rung handles the Alarm Reset Input and Commands
   // and the "Reset and Ack All" Operator Command.
   // This rung processes received Reset Commands from:
   // 1.  The Operator via HMI Operator Command, or
   // 2.  Higher-level strategies via Program Command
   // 3.  Pushbuttons or other block via Input
   // 4.  Resets initiated by other device Operator Commands (if configured to do so)
   // and forwards the Reset to ALL Alarms and latched Shed conditions.
   // The reset starts the Reset Timer (One-Shot Off-Delay)
   // to ensure the output is held on for at least the minimum time.
   // #####  V3.1-00  2014-06-30: Added Not Ready reason bits (Nrdy_xxx)  #####
   // #####  V3.1-01  2014-08-29:  Corrections to Nrdy_ trip and reset logic.  #####
   33: [XIC(OCmd_Reset) OTU(OCmd_Reset) ,[XIC(OCmd_Start) ,XIC(OCmd_Jog) ,XIC(OCmd_Stop) ] XIC(Cfg_OCmdResets) [XIC(Sts_Oper) XIO(Cfg_ProgKeep.1) ,XIC(Sts_Maint) ,XIC(Sts_Prog) XIC(Cfg_OperKeep.1) ] ,XIC(OCmd_ResetAckAll) OTU(OCmd_ResetAckAll) [OTL(PCmd_FailToStartAck) ,OTL(PCmd_FailToStopAck) ,OTL(PCmd_DriveFaultAck) ,OTL(PCmd_IntlkTripAck) ,OTL(PCmd_IOFaultAck) ] ,XIC(PCmd_Reset) [XIC(Cfg_PCmdClear) OTU(PCmd_Reset) ,NOP() ] ,XIC(Inp_Reset) ONS(Wrk_ResetONS) ][OTL(FailToStart.PCmd_Reset) OTL(FailToStop.PCmd_Reset) OTL(IntlkTrip.PCmd_Reset) OTL(IOFault.PCmd_Reset) ,XIC(Sts_FailToStart) RES(Wrk_StartT) ,XIC(Sts_FailToStop) RES(Wrk_StopT) ,OTU(Nrdy_OperPrio) OTU(Nrdy_Fail) ,[XIO(Inp_IOFault) ,XIC(Inp_Sim) ] OTU(Nrdy_IOFault) ,TOF(Wrk_ResetT,?,?) ];
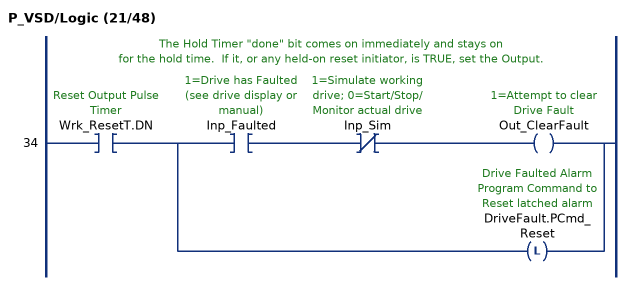
   // The Hold Timer "done" bit comes on immediately and stays on
   // for the hold time.  If it, or any held-on reset initiator, is TRUE, set the Output.
   34: XIC(Wrk_ResetT.DN)[XIC(Inp_Faulted) XIO(Inp_Sim) OTE(Out_ClearFault) ,OTL(DriveFault.PCmd_Reset) ];
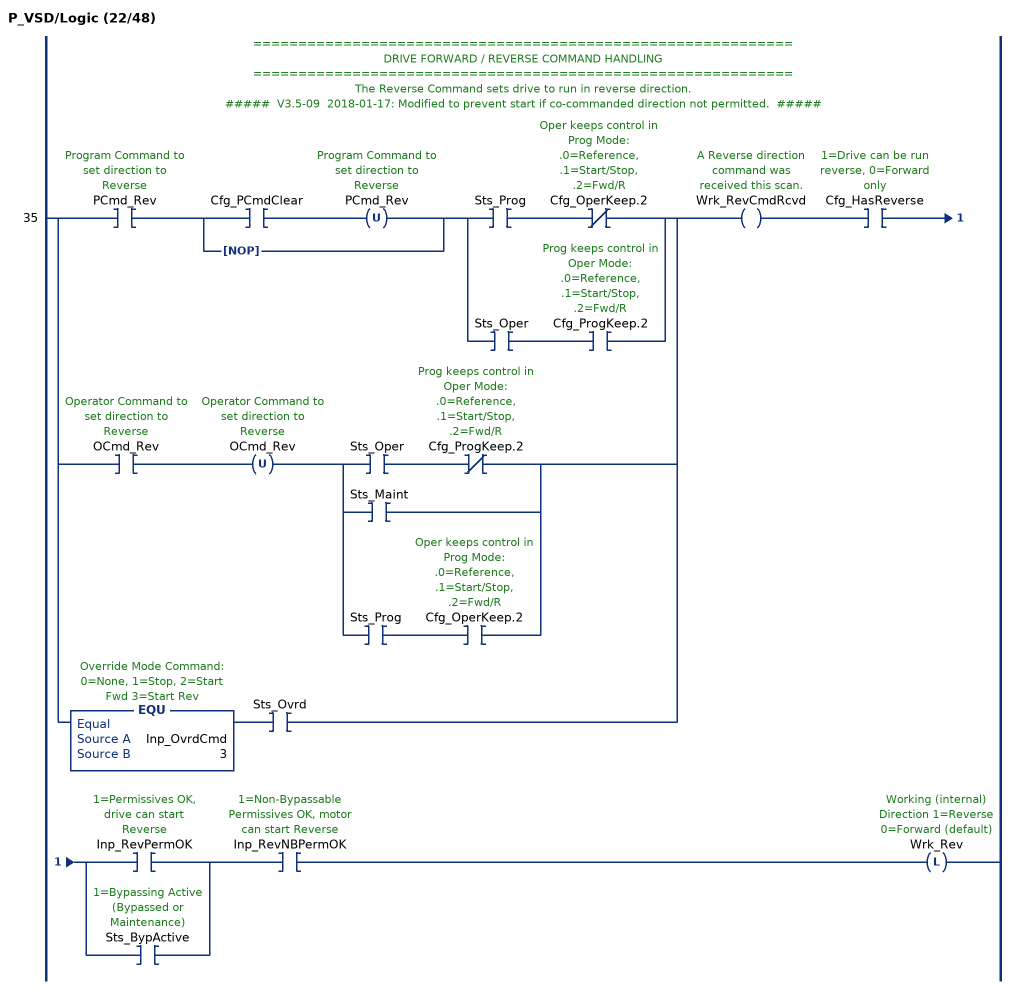
   // ============================================================
   // DRIVE FORWARD / REVERSE COMMAND HANDLING
   // ============================================================
   // The Reverse Command sets drive to run in reverse direction.
   // #####  V3.5-09  2018-01-17: Modified to prevent start if co-commanded direction not permitted.  #####
   35: [XIC(PCmd_Rev) [XIC(Cfg_PCmdClear) OTU(PCmd_Rev) ,NOP() ] [XIC(Sts_Prog) XIO(Cfg_OperKeep.2) ,XIC(Sts_Oper) XIC(Cfg_ProgKeep.2) ] ,XIC(OCmd_Rev) OTU(OCmd_Rev) [XIC(Sts_Oper) XIO(Cfg_ProgKeep.2) ,XIC(Sts_Maint) ,XIC(Sts_Prog) XIC(Cfg_OperKeep.2) ] ,EQU(Inp_OvrdCmd,3) XIC(Sts_Ovrd) ]OTE(Wrk_RevCmdRcvd)XIC(Cfg_HasReverse)[XIC(Inp_RevPermOK) ,XIC(Sts_BypActive) ]XIC(Inp_RevNBPermOK)OTL(Wrk_Rev);
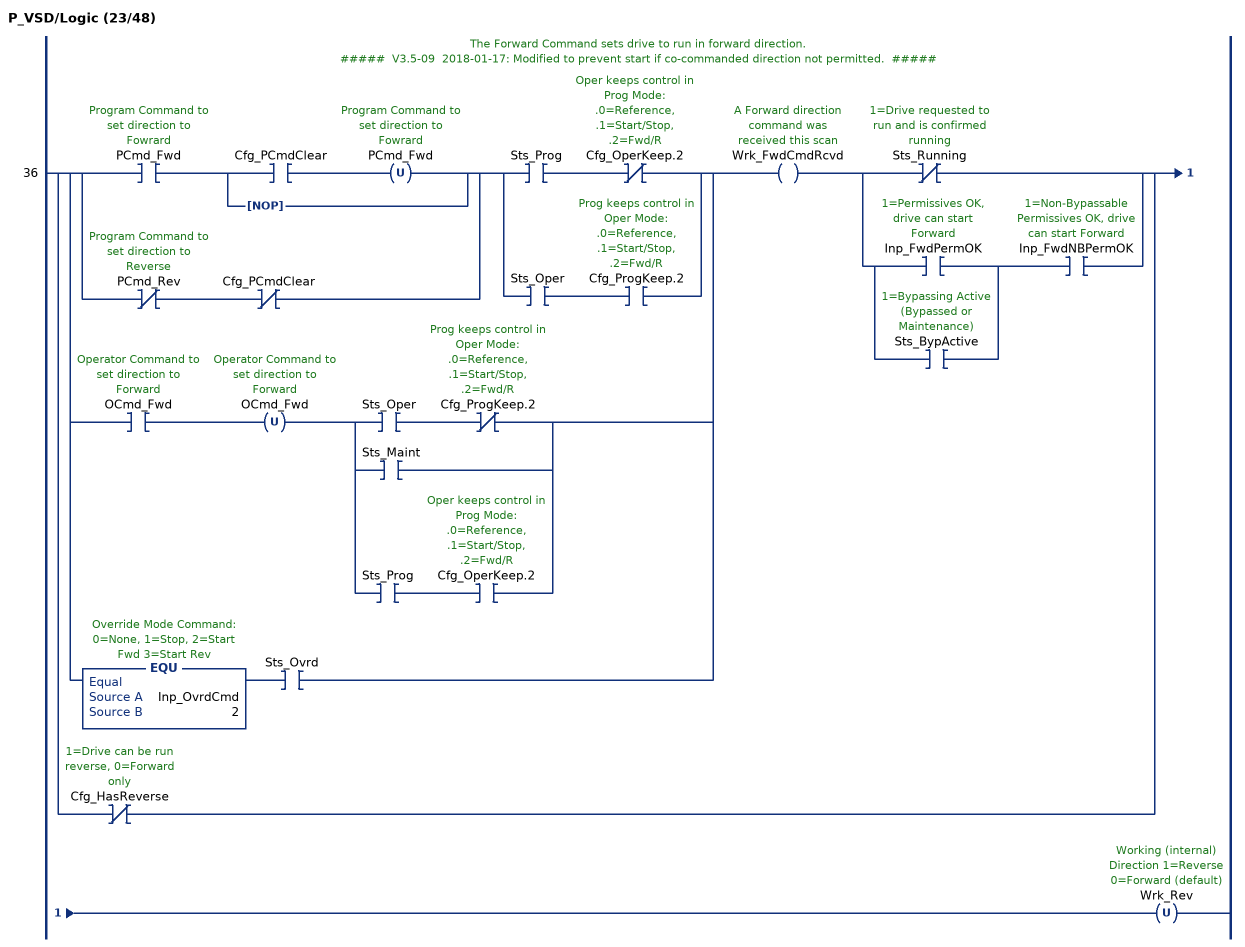
   // The Forward Command sets drive to run in forward direction.
   // #####  V3.5-09  2018-01-17: Modified to prevent start if co-commanded direction not permitted.  #####
   36: [[[XIC(PCmd_Fwd) [XIC(Cfg_PCmdClear) OTU(PCmd_Fwd) ,NOP() ] ,XIO(PCmd_Rev) XIO(Cfg_PCmdClear) ] [XIC(Sts_Prog) XIO(Cfg_OperKeep.2) ,XIC(Sts_Oper) XIC(Cfg_ProgKeep.2) ] ,XIC(OCmd_Fwd) OTU(OCmd_Fwd) [XIC(Sts_Oper) XIO(Cfg_ProgKeep.2) ,XIC(Sts_Maint) ,XIC(Sts_Prog) XIC(Cfg_OperKeep.2) ] ,EQU(Inp_OvrdCmd,2) XIC(Sts_Ovrd) ] OTE(Wrk_FwdCmdRcvd) [XIO(Sts_Running) ,[XIC(Inp_FwdPermOK) ,XIC(Sts_BypActive) ] XIC(Inp_FwdNBPermOK) ] ,XIO(Cfg_HasReverse) ]OTU(Wrk_Rev);
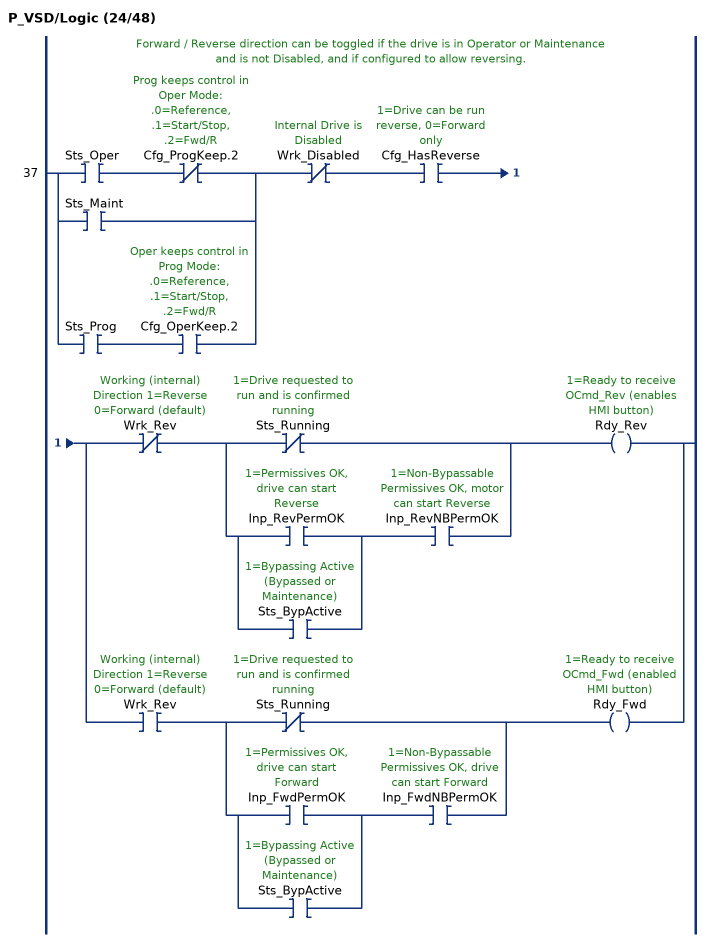
   // Forward / Reverse direction can be toggled if the drive is in Operator or Maintenance
   // and is not Disabled, and if configured to allow reversing.
   37: [XIC(Sts_Oper) XIO(Cfg_ProgKeep.2) ,XIC(Sts_Maint) ,XIC(Sts_Prog) XIC(Cfg_OperKeep.2) ]XIO(Wrk_Disabled)XIC(Cfg_HasReverse)[XIO(Wrk_Rev) [XIO(Sts_Running) ,[XIC(Inp_RevPermOK) ,XIC(Sts_BypActive) ] XIC(Inp_RevNBPermOK) ] OTE(Rdy_Rev) ,XIC(Wrk_Rev) [XIO(Sts_Running) ,[XIC(Inp_FwdPermOK) ,XIC(Sts_BypActive) ] XIC(Inp_FwdNBPermOK) ] OTE(Rdy_Fwd) ];
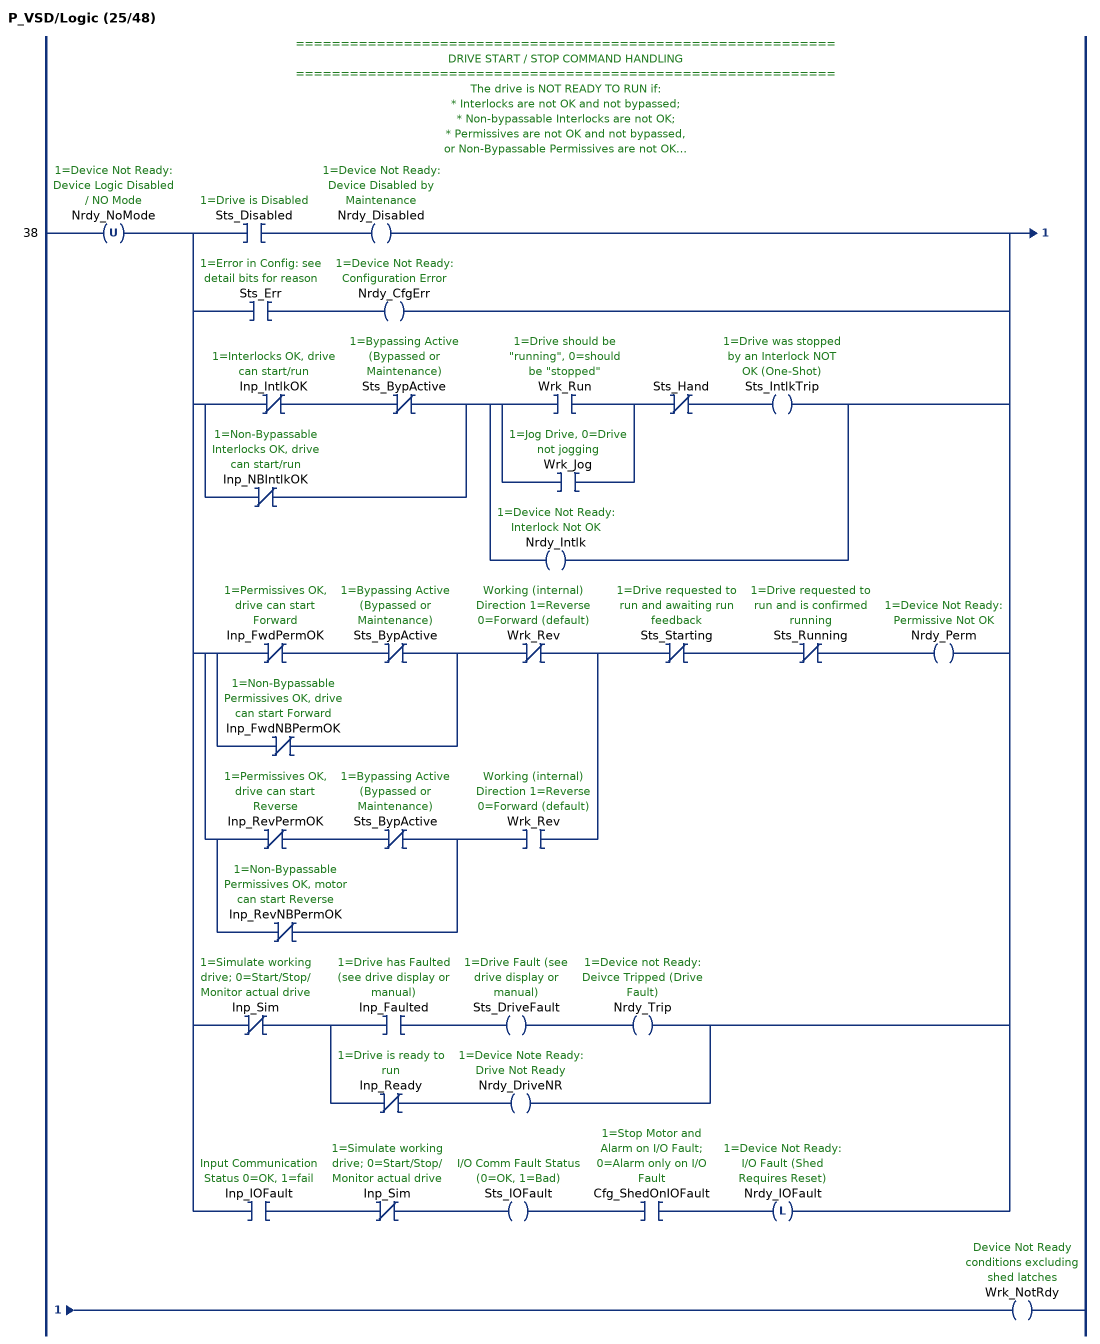
   // ============================================================
   // DRIVE START / STOP COMMAND HANDLING
   // ============================================================
   // The drive is NOT READY TO RUN if:
   // * Interlocks are not OK and not bypassed;
   // * Non-bypassable Interlocks are not OK;
   // * Permissives are not OK and not bypassed,
   // or Non-Bypassable Permissives are not OK,
   // and the motor is not already starting or running;
   // * The drive (not simulated) reports that it is faulted;
   // * There's an I/O failure and the motor is NOT being simulated;
   // * The motor has a Fail to Start that has not been reset;
   // * The drive is disabled (by Maintenance);
   // * This instruction instance has a configuration error.
   // #####  V3.1-00  2014-06-30: Added Not Ready reason bits (Nrdy_xxx)  #####
   // #####  V3.1-01  2014-08-29:  Corrections to Nrdy_ trip and reset logic.  #####
   // #####  V3.5-02  2016-03-22:  Modified to eliminate oscillating Out_Stop on Drive Not Ready.  #####
   // #####  V3.5-09  2018-01-17:  Modified to ensure HAND running shows status RUNNING.  #####
   // #####  Modified to prevent start if co-commanded direction not permitted.  #####
   38: OTU(Nrdy_NoMode)[XIC(Sts_Disabled) OTE(Nrdy_Disabled) ,XIC(Sts_Err) OTE(Nrdy_CfgErr) ,[XIO(Inp_IntlkOK) XIO(Sts_BypActive) ,XIO(Inp_NBIntlkOK) ] [[XIC(Wrk_Run) ,XIC(Wrk_Jog) ] XIO(Sts_Hand) OTE(Sts_IntlkTrip) ,OTE(Nrdy_Intlk) ] ,[[XIO(Inp_FwdPermOK) XIO(Sts_BypActive) ,XIO(Inp_FwdNBPermOK) ] XIO(Wrk_Rev) ,[XIO(Inp_RevPermOK) XIO(Sts_BypActive) ,XIO(Inp_RevNBPermOK) ] XIC(Wrk_Rev) ] XIO(Sts_Starting) XIO(Sts_Running) OTE(Nrdy_Perm) ,XIO(Inp_Sim) [XIC(Inp_Faulted) OTE(Sts_DriveFault) OTE(Nrdy_Trip) ,XIO(Inp_Ready) OTE(Nrdy_DriveNR) ] ,XIC(Inp_IOFault) XIO(Inp_Sim) OTE(Sts_IOFault) XIC(Cfg_ShedOnIOFault) OTL(Nrdy_IOFault) ]OTE(Wrk_NotRdy);
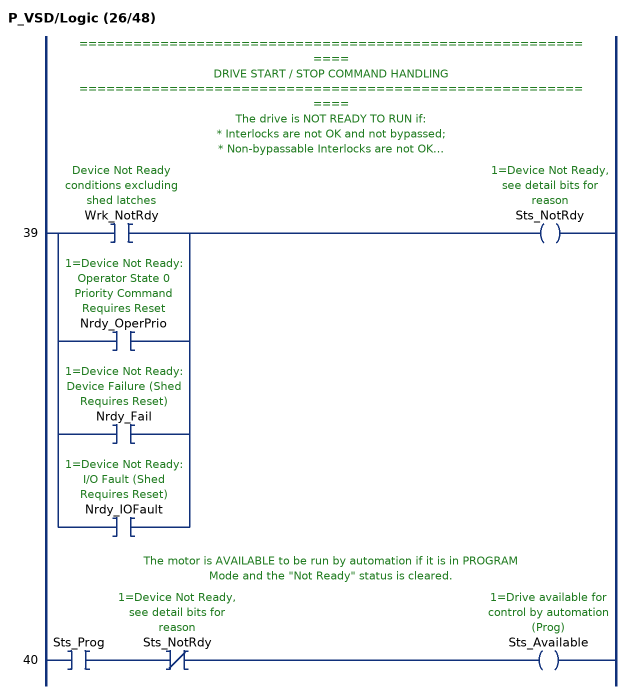
   // ============================================================
   // DRIVE START / STOP COMMAND HANDLING
   // ============================================================
   // The drive is NOT READY TO RUN if:
   // * Interlocks are not OK and not bypassed;
   // * Non-bypassable Interlocks are not OK;
   // * Permissives are not OK and not bypassed,
   // or Non-Bypassable Permissives are not OK,
   // and the motor is not already starting or running;
   // * The drive (not simulated) reports that it is faulted;
   // * There's an I/O failure and the motor is NOT being simulated;
   // * The motor has a Fail to Start that has not been reset;
   // * The drive is disabled (by Maintenance);
   // * This instruction instance has a configuration error.
   // #####  V3.1-00  2014-06-30: Added Not Ready reason bits (Nrdy_xxx)  #####
   // #####  V3.1-01  2014-08-29:  Corrections to Nrdy_ trip and reset logic.  #####
   39: [XIC(Wrk_NotRdy) ,XIC(Nrdy_OperPrio) ,XIC(Nrdy_Fail) ,XIC(Nrdy_IOFault) ]OTE(Sts_NotRdy);
   // The motor is AVAILABLE to be run by automation if it is in PROGRAM
   // Mode and the "Not Ready" status is cleared.
   40: XIC(Sts_Prog)XIO(Sts_NotRdy)OTE(Sts_Available);
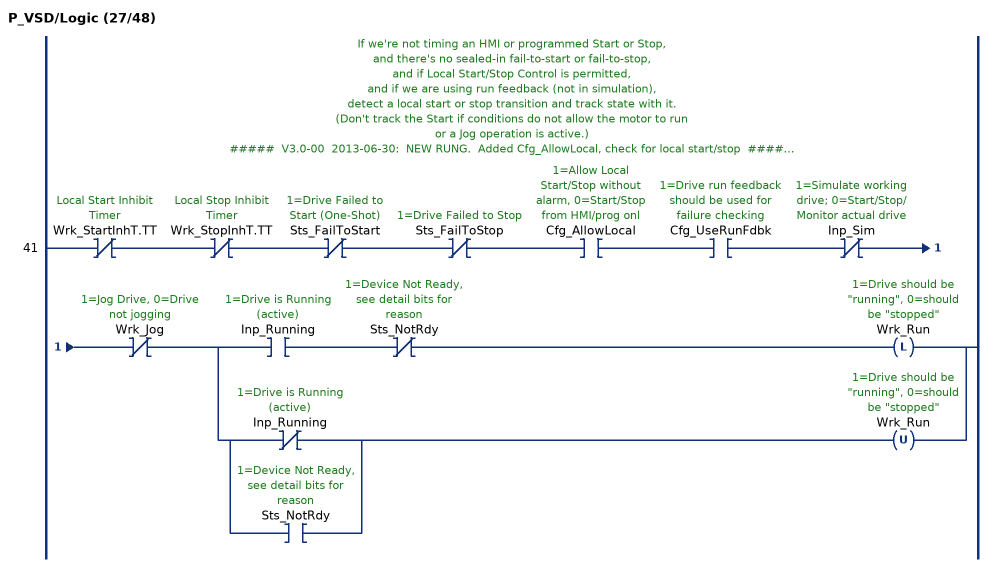
   // If we're not timing an HMI or programmed Start or Stop,
   // and there's no sealed-in fail-to-start or fail-to-stop,
   // and if Local Start/Stop Control is permitted,
   // and if we are using run feedback (not in simulation),
   // detect a local start or stop transition and track state with it.
   // (Don't track the Start if conditions do not allow the motor to run
   // or a Jog operation is active.)
   // #####  V3.0-00  2013-06-30:  NEW RUNG.  Added Cfg_AllowLocal, check for local start/stop  #####
   // #####  V3.1-04 Patch01  2015-09-25:  Modified to correct issue with loss of run feedback.  #####
   // #####  V3.5-04  2016-09-30:  Modified to ignore Jog operation when Local control permitted.  #####
   41: XIO(Wrk_StartInhT.TT)XIO(Wrk_StopInhT.TT)XIO(Sts_FailToStart)XIO(Sts_FailToStop)XIC(Cfg_AllowLocal)XIC(Cfg_UseRunFdbk)XIO(Inp_Sim)XIO(Wrk_Jog)[XIC(Inp_Running) XIO(Sts_NotRdy) OTL(Wrk_Run) ,[XIO(Inp_Running) ,XIC(Sts_NotRdy) ] OTU(Wrk_Run) ];
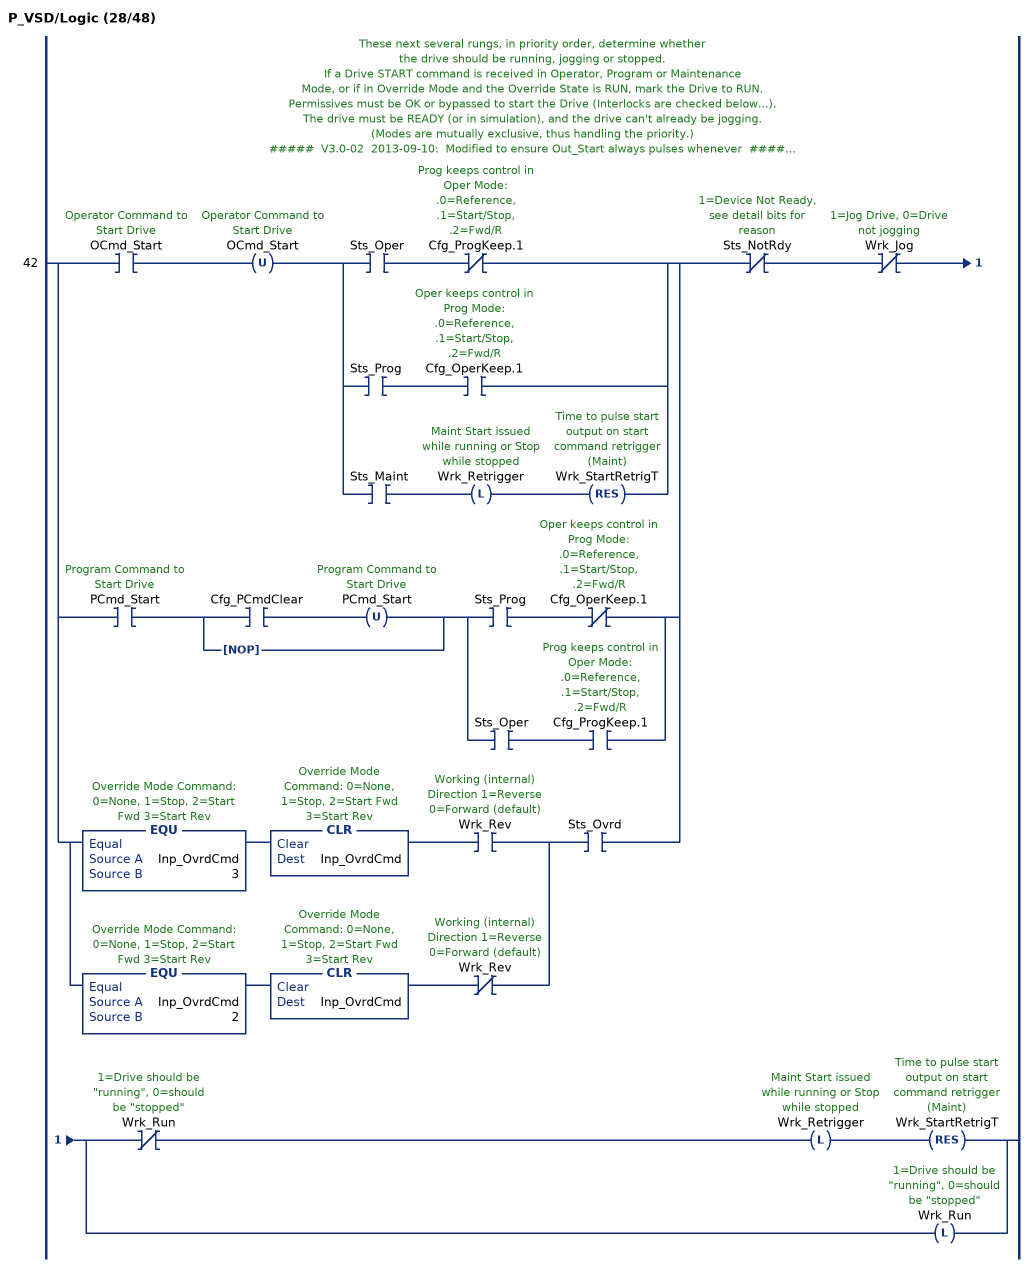
   // These next several rungs, in priority order, determine whether
   // the drive should be running, jogging or stopped.
   // If a Drive START command is received in Operator, Program or Maintenance
   // Mode, or if in Override Mode and the Override State is RUN, mark the Drive to RUN.
   // Permissives must be OK or bypassed to start the Drive (Interlocks are checked below...).
   // The drive must be READY (or in simulation), and the drive can't already be jogging.
   // (Modes are mutually exclusive, thus handling the priority.)
   // #####  V3.0-02  2013-09-10:  Modified to ensure Out_Start always pulses whenever  #####
   // #####  a start command is received, regardless of run feedback state.  #####
   42: [XIC(OCmd_Start) OTU(OCmd_Start) [XIC(Sts_Oper) XIO(Cfg_ProgKeep.1) ,XIC(Sts_Prog) XIC(Cfg_OperKeep.1) ,XIC(Sts_Maint) OTL(Wrk_Retrigger) RES(Wrk_StartRetrigT) ] ,XIC(PCmd_Start) [XIC(Cfg_PCmdClear) OTU(PCmd_Start) ,NOP() ] [XIC(Sts_Prog) XIO(Cfg_OperKeep.1) ,XIC(Sts_Oper) XIC(Cfg_ProgKeep.1) ] ,[EQU(Inp_OvrdCmd,3) CLR(Inp_OvrdCmd) XIC(Wrk_Rev) ,EQU(Inp_OvrdCmd,2) CLR(Inp_OvrdCmd) XIO(Wrk_Rev) ] XIC(Sts_Ovrd) ]XIO(Sts_NotRdy)XIO(Wrk_Jog)[XIO(Wrk_Run) OTL(Wrk_Retrigger) RES(Wrk_StartRetrigT) ,OTL(Wrk_Run) ];
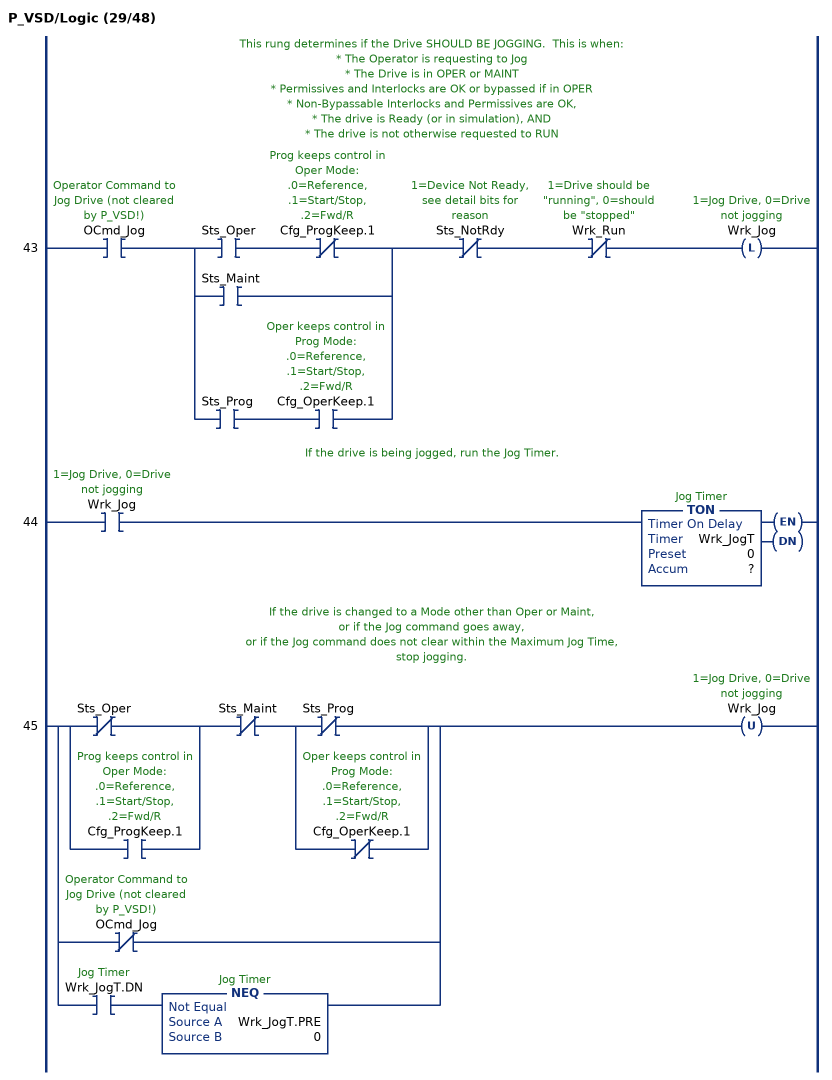
   // This rung determines if the Drive SHOULD BE JOGGING.  This is when:
   // * The Operator is requesting to Jog
   // * The Drive is in OPER or MAINT
   // * Permissives and Interlocks are OK or bypassed if in OPER
   // * Non-Bypassable Interlocks and Permissives are OK,
   // * The drive is Ready (or in simulation), AND
   // * The drive is not otherwise requested to RUN
   43: XIC(OCmd_Jog)[XIC(Sts_Oper) XIO(Cfg_ProgKeep.1) ,XIC(Sts_Maint) ,XIC(Sts_Prog) XIC(Cfg_OperKeep.1) ]XIO(Sts_NotRdy)XIO(Wrk_Run)OTL(Wrk_Jog);
   // If the drive is being jogged, run the Jog Timer.
   44: XIC(Wrk_Jog)TON(Wrk_JogT,?,?);
   // If the drive is changed to a Mode other than Oper or Maint,
   // or if the Jog command goes away,
   // or if the Jog command does not clear within the Maximum Jog Time,
   // stop jogging.
   45: [[XIO(Sts_Oper) ,XIC(Cfg_ProgKeep.1) ] XIO(Sts_Maint) [XIO(Sts_Prog) ,XIO(Cfg_OperKeep.1) ] ,XIO(OCmd_Jog) ,XIC(Wrk_JogT.DN) NEQ(Wrk_JogT.PRE,0) ]OTU(Wrk_Jog);
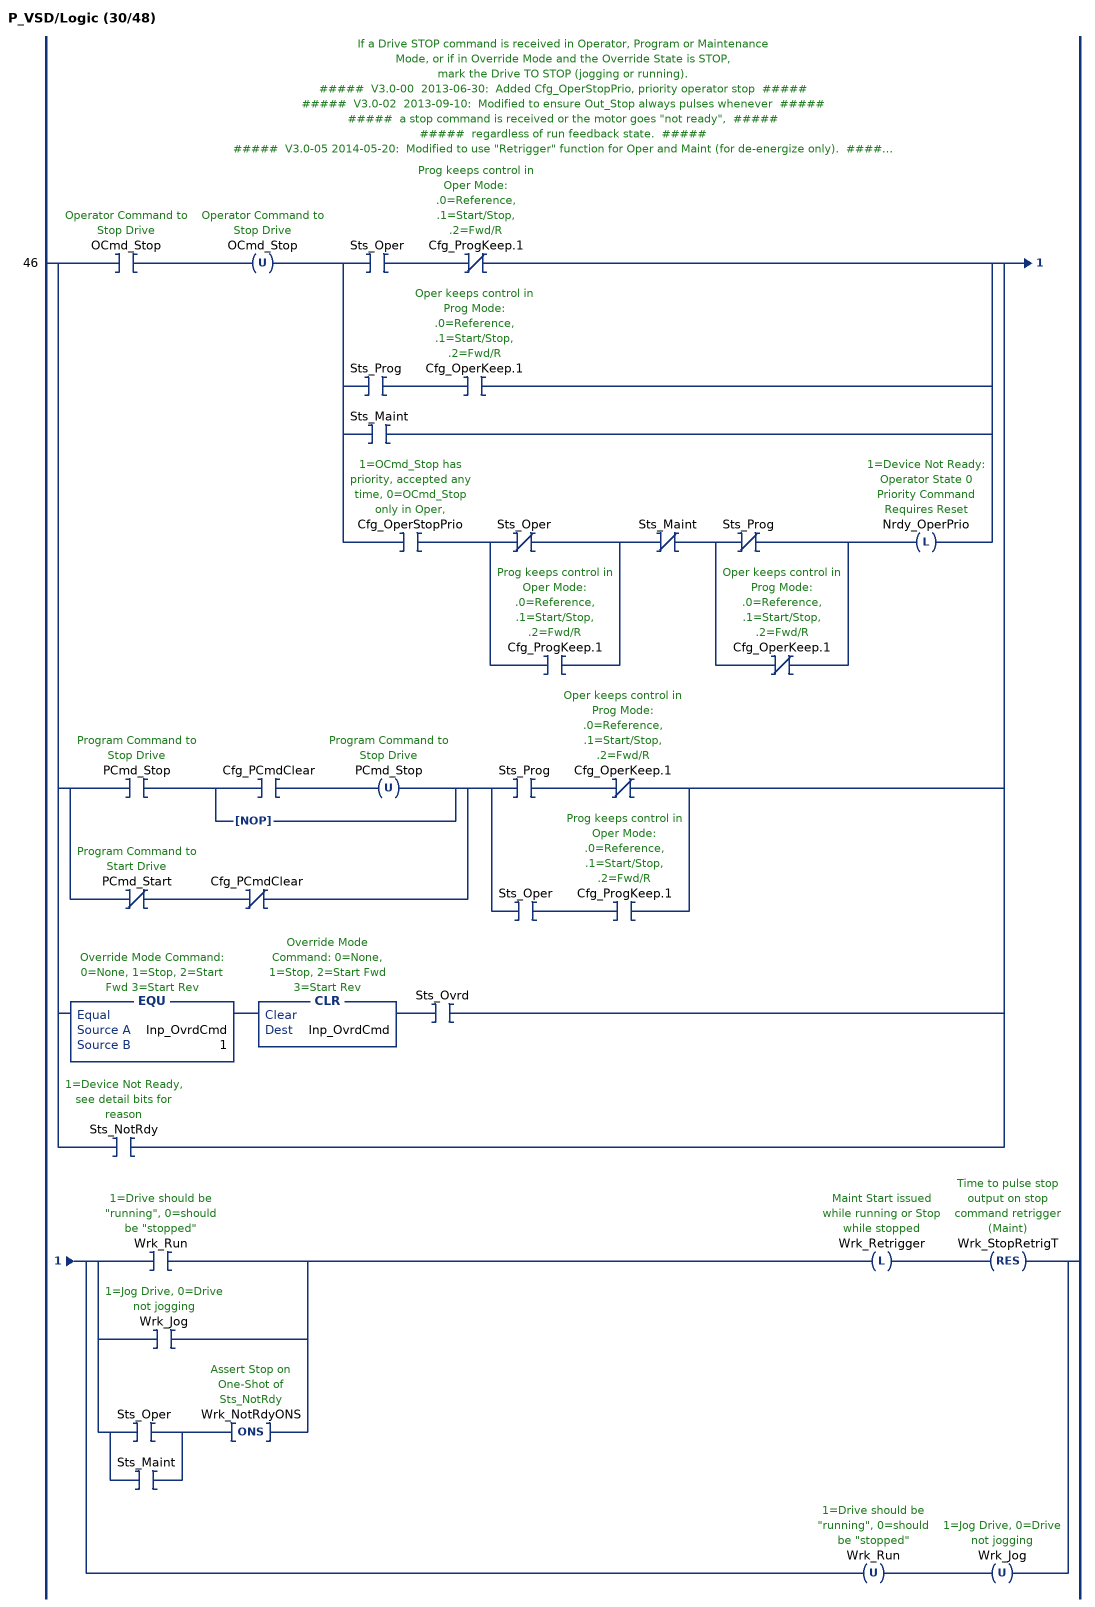
   // If a Drive STOP command is received in Operator, Program or Maintenance
   // Mode, or if in Override Mode and the Override State is STOP,
   // mark the Drive TO STOP (jogging or running).
   // #####  V3.0-00  2013-06-30:  Added Cfg_OperStopPrio, priority operator stop  #####
   // #####  V3.0-02  2013-09-10:  Modified to ensure Out_Stop always pulses whenever  #####
   // #####  a stop command is received or the motor goes "not ready",  #####
   // #####  regardless of run feedback state.  #####
   // #####  V3.0-05 2014-05-20:  Modified to use "Retrigger" function for Oper and Maint (for de-energize only).  #####
   // #####  V3.0-06 2014-06-12:  Modified to use "Retrigger" function for Oper and Maint (for de-energize only).  #####
   // #####  V3.0-07 2014-06-30:  Modified to one-shot assert stop retrigger on Not Ready status.  #####
   // #####  V3.1-00  2014-06-30: Added Not Ready reason bits (Nrdy_xxx)  #####
   // #####  V3.1-03  2015-01-16:   Modified stop retriggering to handle asynchronous Prog mode owner.  #####
   46: [XIC(OCmd_Stop) OTU(OCmd_Stop) [XIC(Sts_Oper) XIO(Cfg_ProgKeep.1) ,XIC(Sts_Prog) XIC(Cfg_OperKeep.1) ,XIC(Sts_Maint) ,XIC(Cfg_OperStopPrio) [XIO(Sts_Oper) ,XIC(Cfg_ProgKeep.1) ] XIO(Sts_Maint) [XIO(Sts_Prog) ,XIO(Cfg_OperKeep.1) ] OTL(Nrdy_OperPrio) ] ,[XIC(PCmd_Stop) [XIC(Cfg_PCmdClear) OTU(PCmd_Stop) ,NOP() ] ,XIO(PCmd_Start) XIO(Cfg_PCmdClear) ] [XIC(Sts_Prog) XIO(Cfg_OperKeep.1) ,XIC(Sts_Oper) XIC(Cfg_ProgKeep.1) ] ,EQU(Inp_OvrdCmd,1) CLR(Inp_OvrdCmd) XIC(Sts_Ovrd) ,XIC(Sts_NotRdy) ][[XIC(Wrk_Run) ,XIC(Wrk_Jog) ,[XIC(Sts_Oper) ,XIC(Sts_Maint) ] ONS(Wrk_NotRdyONS) ] OTL(Wrk_Retrigger) RES(Wrk_StopRetrigT) ,OTU(Wrk_Run) OTU(Wrk_Jog) ];
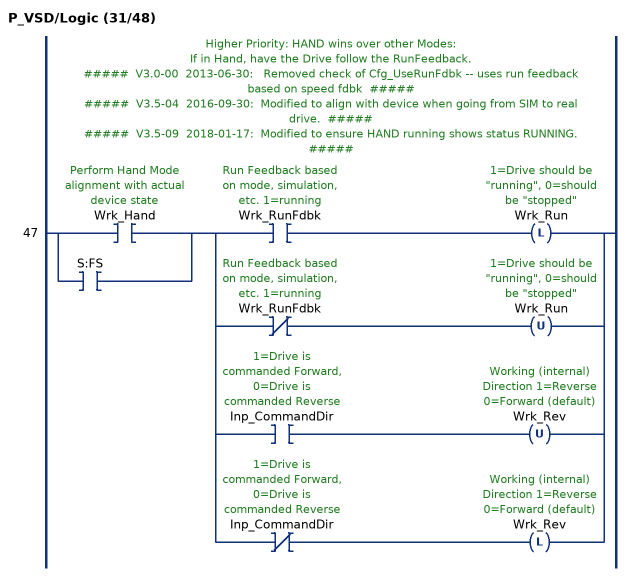
   // Higher Priority: HAND wins over other Modes:
   // If in Hand, have the Drive follow the RunFeedback.
   // #####  V3.0-00  2013-06-30:   Removed check of Cfg_UseRunFdbk -- uses run feedback  based on speed fdbk  #####
   // #####  V3.5-04  2016-09-30:  Modified to align with device when going from SIM to real drive.  #####
   // #####  V3.5-09  2018-01-17:  Modified to ensure HAND running shows status RUNNING.  #####
   47: [XIC(Wrk_Hand) ,XIC(S:FS) ][XIC(Wrk_RunFdbk) OTL(Wrk_Run) ,XIO(Wrk_RunFdbk) OTU(Wrk_Run) ,XIC(Inp_CommandDir) OTU(Wrk_Rev) ,XIO(Inp_CommandDir) OTL(Wrk_Rev) ];
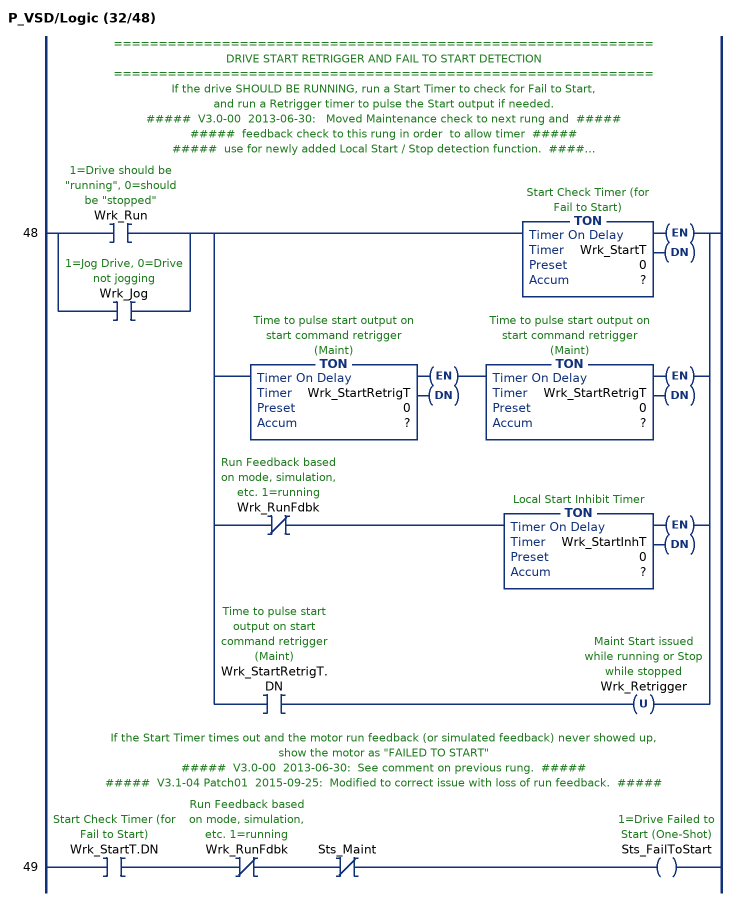
   // ============================================================
   // DRIVE START RETRIGGER AND FAIL TO START DETECTION
   // ============================================================
   // If the drive SHOULD BE RUNNING, run a Start Timer to check for Fail to Start,
   //  and run a Retrigger timer to pulse the Start output if needed.
   // #####  V3.0-00  2013-06-30:   Moved Maintenance check to next rung and  #####
   // #####  feedback check to this rung in order  to allow timer  #####
   // #####  use for newly added Local Start / Stop detection function.  #####
   // #####  V3.1-04 Patch01  2015-09-25:  Modified to correct issue with loss of run feedback.  #####
   // @@@@@  The TON on the second branch is doubled to ensure it goes  @@@@@
   // @@@@@  the same scan it is enabled if its preset is zero.  @@@@@
   48: [XIC(Wrk_Run) ,XIC(Wrk_Jog) ][TON(Wrk_StartT,?,?) ,TON(Wrk_StartRetrigT,?,?) TON(Wrk_StartRetrigT,?,?) ,XIO(Wrk_RunFdbk) TON(Wrk_StartInhT,?,?) ,XIC(Wrk_StartRetrigT.DN) OTU(Wrk_Retrigger) ];
   // If the Start Timer times out and the motor run feedback (or simulated feedback) never showed up,
   // show the motor as "FAILED TO START"
   // #####  V3.0-00  2013-06-30:  See comment on previous rung.  #####
   // #####  V3.1-04 Patch01  2015-09-25:  Modified to correct issue with loss of run feedback.  #####
   49: XIC(Wrk_StartT.DN)XIO(Wrk_RunFdbk)XIO(Sts_Maint)OTE(Sts_FailToStart);
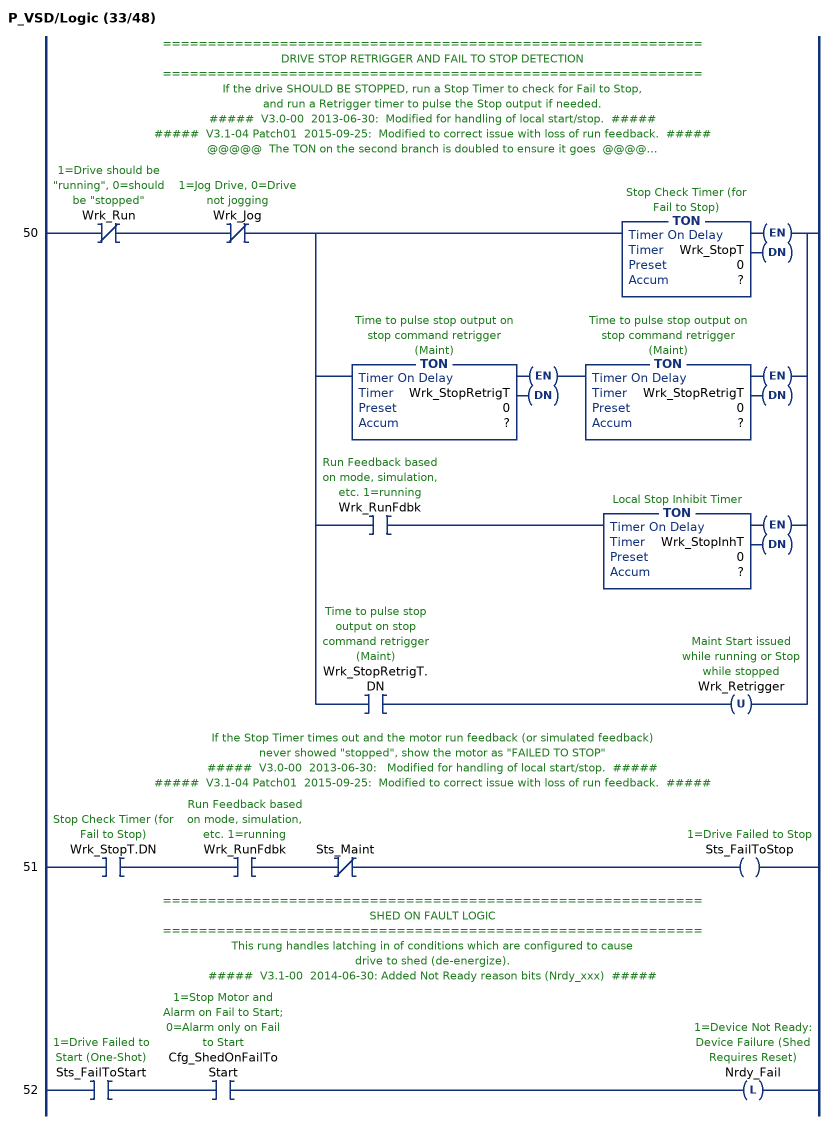
   // ============================================================
   // DRIVE STOP RETRIGGER AND FAIL TO STOP DETECTION
   // ============================================================
   // If the drive SHOULD BE STOPPED, run a Stop Timer to check for Fail to Stop,
   //  and run a Retrigger timer to pulse the Stop output if needed.
   // #####  V3.0-00  2013-06-30:  Modified for handling of local start/stop.  #####
   // #####  V3.1-04 Patch01  2015-09-25:  Modified to correct issue with loss of run feedback.  #####
   // @@@@@  The TON on the second branch is doubled to ensure it goes  @@@@@
   // @@@@@  true the same scan it is enabled if its preset is zero.  @@@@@
   50: XIO(Wrk_Run)XIO(Wrk_Jog)[TON(Wrk_StopT,?,?) ,TON(Wrk_StopRetrigT,?,?) TON(Wrk_StopRetrigT,?,?) ,XIC(Wrk_RunFdbk) TON(Wrk_StopInhT,?,?) ,XIC(Wrk_StopRetrigT.DN) OTU(Wrk_Retrigger) ];
   // If the Stop Timer times out and the motor run feedback (or simulated feedback)
   // never showed "stopped", show the motor as "FAILED TO STOP"
   // #####  V3.0-00  2013-06-30:   Modified for handling of local start/stop.  #####
   // #####  V3.1-04 Patch01  2015-09-25:  Modified to correct issue with loss of run feedback.  #####
   51: XIC(Wrk_StopT.DN)XIC(Wrk_RunFdbk)XIO(Sts_Maint)OTE(Sts_FailToStop);
   // ============================================================
   // SHED ON FAULT LOGIC
   // ============================================================
   // This rung handles latching in of conditions which are configured to cause
   // drive to shed (de-energize).
   // #####  V3.1-00  2014-06-30: Added Not Ready reason bits (Nrdy_xxx)  #####
   52: XIC(Sts_FailToStart)XIC(Cfg_ShedOnFailToStart)OTL(Nrdy_Fail);
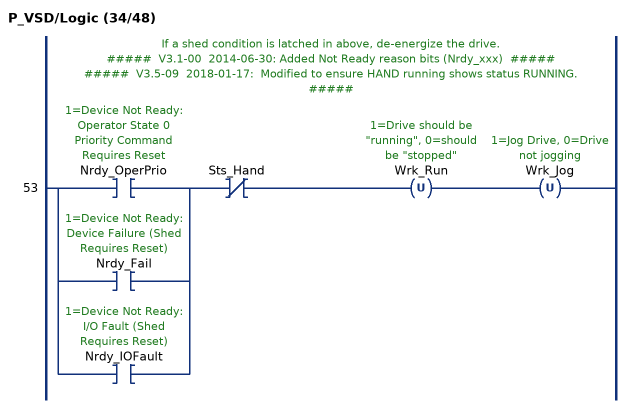
   // If a shed condition is latched in above, de-energize the drive.
   // #####  V3.1-00  2014-06-30: Added Not Ready reason bits (Nrdy_xxx)  #####
   // #####  V3.5-09  2018-01-17:  Modified to ensure HAND running shows status RUNNING.  #####
   53: [XIC(Nrdy_OperPrio) ,XIC(Nrdy_Fail) ,XIC(Nrdy_IOFault) ]XIO(Sts_Hand)OTU(Wrk_Run)OTU(Wrk_Jog);
